C07288=1034.906,183.861,395.226,169.883,42.558,158.045
C07289=1034.912,184.110,395.201,169.886,42.558,158.045
C07290=1034.918,184.359,395.178,169.889,42.558,158.045
C07291=1034.925,184.608,395.155,169.892,42.557,158.046
C07292=1034.930,184.857,395.130,169.895,42.557,158.046
C07293=1034.936,185.105,395.107,169.898,42.556,158.046
C07294=1034.942,185.355,395.082,169.901,42.556,158.046
C07295=1034.948,185.603,395.058,169.904,42.555,158.046
C07296=1034.954,185.852,395.034,169.907,42.555,158.046
C07297=1034.960,186.100,395.010,169.911,42.555,158.046
C07298=1034.966,186.350,394.985,169.914,42.554,158.046
C07299=1034.972,186.598,394.962,169.917,42.554,158.047
C07300=1034.977,186.847,394.937,169.920,42.553,158.047
C07301=1034.984,187.095,394.913,169.923,42.553,158.047
C07302=1034.990,187.344,394.890,169.926,42.552,158.047
C07303=1034.996,187.593,394.865,169.929,42.552,158.047
C07304=1035.002,187.841,394.842,169.932,42.552,158.047
C07305=1035.008,188.091,394.817,169.935,42.552,158.047
C07306=1035.014,188.339,394.793,169.938,42.551,158.048
C07307=1035.021,188.624,394.766,169.941,42.551,158.048
C07308=1035.028,188.907,394.738,169.944,42.550,158.048
C07309=1035.035,189.191,394.710,169.948,42.550,158.048
C07310=1035.041,189.476,394.683,169.952,42.550,158.048
C07311=1035.047,189.724,394.659,169.955,42.549,158.048
C07312=1035.053,189.973,394.635,169.958,42.549,158.048
C07313=1035.059,190.222,394.609,169.962,42.548,158.049
C07314=1035.066,190.470,394.586,169.965,42.548,158.049
C07315=1035.071,190.719,394.561,169.968,42.547,158.049
C07316=1035.077,190.968,394.538,169.971,42.547,158.049
C07317=1035.083,191.217,394.513,169.974,42.547,158.049
C07318=1035.089,191.465,394.489,169.977,42.546,158.049
C07319=1035.095,191.715,394.465,169.980,42.546,158.049
C07320=1035.102,191.964,394.441,169.983,42.545,158.050
C07321=1035.108,192.212,394.416,169.986,42.546,158.050
C07322=1035.114,192.460,394.392,169.989,42.545,158.050
C07323=1035.119,192.709,394.367,169.992,42.545,158.050
C07324=1035.126,192.958,394.343,169.996,42.544,158.050
C07325=1035.132,193.207,394.319,169.999,42.544,158.050
C07326=1035.138,193.455,394.294,170.002,42.544,158.050
C07327=1035.144,193.704,394.270,170.006,42.543,158.051
C07328=1035.151,193.953,394.246,170.009,42.543,158.051
C07329=1035.156,194.202,394.221,170.012,42.542,158.051
C07330=1035.163,194.450,394.197,170.015,42.542,158.051
C07331=1035.169,194.700,394.172,170.018,42.542,158.051
C07332=1035.175,194.948,394.148,170.021,42.541,158.051
C07333=1035.181,195.196,394.123,170.024,42.541,158.051
C07334=1035.188,195.445,394.099,170.027,42.540,158.052
C07335=1035.193,195.694,394.075,170.031,42.541,158.052
C07336=1035.200,195.942,394.050,170.035,42.540,158.052
C07337=1035.206,196.192,394.025,170.038,42.540,158.052
C07338=1035.212,196.440,394.002,170.041,42.539,158.052
C07339=1035.218,196.689,393.976,170.044,42.539,158.052
C07340=1035.224,196.938,393.952,170.047,42.539,158.053
C07341=1035.231,197.187,393.928,170.050,42.538,158.053
C07342=1035.236,197.435,393.903,170.053,42.538,158.053
C07343=1035.243,197.684,393.879,170.057,42.538,158.053
C07344=1035.249,197.932,393.853,170.060,42.537,158.053
C07345=1035.256,198.181,393.829,170.063,42.537,158.053
C07346=1035.262,198.429,393.804,170.067,42.537,158.054
C07347=1035.268,198.678,393.780,170.070,42.536,158.054
C07348=1035.274,198.927,393.755,170.073,42.536,158.054
C07349=1035.281,199.176,393.731,170.077,42.536,158.054
C07350=1035.287,199.425,393.706,170.080,42.536,158.054
C07351=1035.293,199.673,393.682,170.083,42.535,158.054
C07352=1035.299,199.922,393.657,170.086,42.535,158.054
C07353=1035.305,200.171,393.632,170.089,42.535,158.055
C07354=1035.312,200.419,393.607,170.092,42.534,158.055
C07355=1035.318,200.669,393.583,170.096,42.534,158.055
C07356=1035.325,200.916,393.558,170.100,42.534,158.055
C07357=1035.330,201.166,393.534,170.103,42.533,158.055
C07358=1035.337,201.414,393.508,170.106,42.533,158.056
C07359=1035.343,201.663,393.483,170.109,42.533,158.056
C07360=1035.349,201.912,393.458,170.112,42.533,158.056
C07361=1035.354,202.160,393.433,170.116,42.532,158.056
C07362=1035.361,202.409,393.408,170.119,42.533,158.056
C07363=1035.367,202.657,393.383,170.122,42.532,158.057
C07364=1035.373,202.907,393.358,170.126,42.532,158.057
C07365=1035.380,203.155,393.333,170.129,42.532,158.057
C07366=1035.386,203.404,393.308,170.133,42.532,158.057
C07367=1035.391,203.652,393.283,170.136,42.532,158.057
C07368=1035.397,203.901,393.258,170.139,42.532,158.058
C07369=1035.404,204.150,393.233,170.142,42.532,158.058
C07370=1035.410,204.398,393.208,170.145,42.531,158.058
C07371=1035.436,205.448,393.102,170.465,42.636,158.102
C07372=1035.445,205.782,393.066,170.469,42.636,158.102
C07373=1035.454,206.115,393.031,170.472,42.637,158.103
C07374=1035.463,206.448,392.995,170.475,42.638,158.103
C07375=1035.472,206.782,392.960,170.478,42.639,158.104
C07376=1035.479,207.030,392.934,170.480,42.639,158.104
C07377=1035.486,207.279,392.907,170.483,42.640,158.104
C07378=1035.493,207.528,392.881,170.486,42.640,158.105
C07379=1035.499,207.776,392.854,170.488,42.641,158.105
C07380=1035.506,208.025,392.828,170.491,42.641,158.105
C07381=1035.512,208.273,392.802,170.493,42.642,158.105
C07382=1035.519,208.522,392.775,170.495,42.643,158.106
C07383=1035.526,208.771,392.748,170.498,42.644,158.106
C07384=1035.532,209.019,392.722,170.500,42.644,158.106
C07385=1035.540,209.267,392.695,170.502,42.645,158.107
C07386=1035.546,209.516,392.668,170.505,42.645,158.107
C07387=1035.553,209.764,392.642,170.508,42.646,158.107
C07388=1035.560,210.013,392.616,170.510,42.646,158.108
C07389=1035.566,210.262,392.589,170.513,42.647,158.108
C07390=1035.573,210.509,392.562,170.515,42.647,158.108
C07391=1035.580,210.758,392.535,170.517,42.648,158.108
C07392=1035.586,211.007,392.508,170.520,42.649,158.109
C07393=1035.593,211.255,392.482,170.522,42.650,158.109
C07394=1035.600,211.504,392.456,170.524,42.650,158.109
C07395=1035.607,211.752,392.428,170.528,42.651,158.110
C07396=1035.613,212.000,392.402,170.530,42.651,158.110
C07397=1035.620,212.249,392.375,170.532,42.652,158.110
C07398=1035.627,212.497,392.348,170.535,42.653,158.111
C07399=1035.633,212.746,392.321,170.537,42.653,158.111
C07400=1035.639,212.995,392.294,170.539,42.654,158.111
C07401=1035.647,213.243,392.267,170.542,42.654,158.111
C07402=1035.652,213.491,392.240,170.545,42.655,158.112
C07403=1035.660,213.740,392.214,170.547,42.656,158.112
C07404=1035.666,213.989,392.186,170.550,42.656,158.112
C07405=1035.673,214.237,392.160,170.552,42.657,158.113
C07406=1035.679,214.485,392.133,170.554,42.658,158.113
C07407=1035.687,214.734,392.106,170.557,42.659,158.113
C07408=1035.693,214.983,392.079,170.559,42.659,158.114
C07409=1035.700,215.230,392.052,170.562,42.660,158.114
C07410=1035.706,215.479,392.025,170.565,42.660,158.114
C07411=1035.714,215.727,391.998,170.567,42.661,158.115
C07412=1035.719,215.976,391.972,170.569,42.662,158.115
C07413=1035.727,216.224,391.944,170.572,42.662,158.115
C07414=1035.733,216.473,391.917,170.575,42.663,158.116
C07415=1035.741,216.721,391.890,170.577,42.663,158.116
C07416=1035.747,216.970,391.863,170.580,42.664,158.116
C07417=1035.754,217.218,391.836,170.582,42.664,158.116
C07418=1035.760,217.467,391.809,170.584,42.665,158.117
C07419=1035.767,217.715,391.782,170.588,42.666,158.117
C07420=1035.774,217.964,391.755,170.590,42.666,158.117
C07421=1035.781,218.212,391.728,170.593,42.667,158.118
C07422=1035.787,218.460,391.702,170.595,42.668,158.118
C07423=1035.794,218.709,391.674,170.597,42.669,158.118
C07424=1035.801,218.958,391.647,170.600,42.669,158.119
C07425=1035.808,219.206,391.620,170.603,42.670,158.119
C07426=1035.815,219.455,391.593,170.605,42.670,158.119
C07427=1035.821,219.702,391.566,170.608,42.671,158.120
C07428=1035.831,220.042,391.528,170.611,42.672,158.120
C07429=1035.839,220.381,391.492,170.614,42.672,158.120
C07430=1035.848,220.720,391.454,170.618,42.674,158.121
C07431=1035.857,221.059,391.417,170.621,42.675,158.121
C07432=1035.864,221.308,391.390,170.625,42.675,158.122
C07433=1035.870,221.556,391.362,170.627,42.676,158.122
C07434=1035.876,221.804,391.334,170.630,42.677,158.122
C07435=1035.884,222.052,391.307,170.632,42.678,158.123
C07436=1035.890,222.301,391.280,170.635,42.678,158.123
C07437=1035.897,222.550,391.253,170.638,42.679,158.123
C07438=1035.904,222.798,391.225,170.640,42.680,158.124
C07439=1035.910,223.047,391.197,170.642,42.680,158.124
C07440=1035.917,223.296,391.170,170.646,42.681,158.124
C07441=1035.923,223.543,391.143,170.648,42.681,158.125
C07442=1035.930,223.791,391.116,170.650,42.682,158.125
C07443=1035.937,224.040,391.088,170.653,42.683,158.125
C07444=1035.944,224.288,391.060,170.656,42.683,158.126
C07445=1035.950,224.537,391.032,170.659,42.684,158.126
C07446=1035.957,224.786,391.006,170.661,42.685,158.126
C07447=1035.964,225.034,390.978,170.663,42.686,158.127
C07448=1035.971,225.282,390.951,170.667,42.686,158.127
C07449=1035.977,225.531,390.923,170.669,42.687,158.127
C07450=1035.984,225.779,390.895,170.671,42.688,158.128
C07451=1035.990,226.027,390.868,170.675,42.688,158.128
C07452=1035.998,226.275,390.841,170.677,42.689,158.128
C07453=1036.004,226.524,390.813,170.680,42.690,158.129
C07454=1036.011,226.772,390.785,170.682,42.690,158.129
C07455=1036.017,227.021,390.758,170.685,42.691,158.129
C07456=1036.024,227.270,390.730,170.688,42.692,158.130
C07457=1036.031,227.518,390.703,170.690,42.692,158.130
C07458=1036.037,227.766,390.675,170.693,42.693,158.130
C07459=1036.045,228.015,390.648,170.696,42.694,158.131
C07460=1036.051,228.263,390.620,170.698,42.694,158.131
C07461=1036.058,228.511,390.592,170.701,42.695,158.131
C07462=1036.065,228.760,390.565,170.704,42.696,158.132
C07463=1036.071,229.008,390.536,170.706,42.696,158.132
C07464=1036.078,229.256,390.508,170.710,42.697,158.132
C07465=1036.084,229.505,390.480,170.712,42.698,158.133
C07466=1036.091,229.753,390.452,170.714,42.698,158.133
C07467=1036.098,230.002,390.425,170.717,42.699,158.134
C07468=1036.104,230.250,390.397,170.720,42.699,158.134
C07469=1036.111,230.499,390.369,170.722,42.700,158.134
C07470=1036.118,230.747,390.341,170.725,42.701,158.135
C07471=1036.124,230.996,390.314,170.728,42.702,158.135
C07472=1036.131,231.243,390.285,170.731,42.702,158.135
C07473=1036.138,231.492,390.258,170.733,42.703,158.136
C07474=1036.145,231.740,390.230,170.736,42.704,158.136
C07475=1036.151,231.989,390.201,170.739,42.705,158.136
C07476=1036.157,232.237,390.174,170.741,42.706,158.137
C07477=1036.164,232.485,390.145,170.745,42.706,158.137
C07478=1036.171,232.734,390.118,170.747,42.707,158.137
C07479=1036.178,232.982,390.090,170.749,42.708,158.138
C07480=1036.184,233.230,390.061,170.753,42.709,158.138
C07481=1036.191,233.479,390.033,170.755,42.710,158.138
C07482=1036.197,233.727,390.005,170.759,42.710,158.139
C07483=1036.204,233.976,389.978,170.761,42.711,158.139
C07484=1036.213,234.307,389.939,170.765,42.712,158.140
C07485=1036.222,234.639,389.903,170.768,42.713,158.140
C07486=1036.230,234.970,389.864,170.772,42.714,158.141
C07487=1036.240,235.301,389.827,170.776,42.715,158.141
C07488=1036.246,235.550,389.799,170.779,42.716,158.141
C07489=1036.252,235.798,389.771,170.781,42.717,158.142
C07490=1036.259,236.046,389.742,170.784,42.717,158.142
C07491=1036.266,236.295,389.714,170.787,42.718,158.142
C07492=1036.273,236.543,389.686,170.789,42.719,158.143
C07493=1036.279,236.792,389.657,170.793,42.719,158.143
C07494=1036.286,237.040,389.630,170.795,42.720,158.144
C07495=1036.293,237.288,389.601,170.798,42.721,158.144
C07496=1036.300,237.537,389.574,170.801,42.722,158.144
C07497=1036.306,237.785,389.545,170.803,42.723,158.145
C07498=1036.313,238.033,389.517,170.806,42.723,158.145
C07499=1036.320,238.281,389.488,170.809,42.724,158.145
C07500=1036.326,238.530,389.460,170.812,42.725,158.146
C07501=1036.333,238.778,389.431,170.815,42.726,158.146
C07502=1036.340,239.027,389.403,170.818,42.726,158.147
C07503=1036.347,239.275,389.375,170.821,42.727,158.147
C07504=1036.353,239.523,389.347,170.823,42.728,158.147
C07505=1036.360,239.771,389.318,170.826,42.728,158.148
C07506=1036.367,240.020,389.289,170.829,42.729,158.148
C07507=1036.373,240.268,389.261,170.832,42.730,158.148
C07508=1036.380,240.516,389.233,170.835,42.731,158.149
C07509=1036.387,240.765,389.205,170.838,42.732,158.149
C07510=1036.393,241.013,389.176,170.841,42.732,158.150
C07511=1036.400,241.261,389.147,170.843,42.733,158.150
C07512=1036.407,241.509,389.118,170.846,42.734,158.150
C07513=1036.413,241.758,389.090,170.849,42.735,158.151
C07514=1036.420,242.006,389.061,170.852,42.736,158.151
C07515=1036.426,242.254,389.032,170.855,42.737,158.151
C07516=1036.433,242.503,389.005,170.858,42.737,158.152
C07517=1036.440,242.751,388.975,170.861,42.738,158.152
C07518=1036.447,242.999,388.947,170.864,42.739,158.153
C07519=1036.453,243.247,388.918,170.866,42.740,158.153
C07520=1036.459,243.495,388.889,170.869,42.741,158.153
C07521=1036.466,243.744,388.861,170.872,42.742,158.154
C07522=1036.473,243.993,388.831,170.875,42.743,158.154
C07523=1036.480,244.241,388.803,170.878,42.743,158.155
C07524=1036.486,244.489,388.774,170.881,42.744,158.155
C07525=1036.493,244.737,388.746,170.884,42.745,158.155
C07526=1036.499,244.985,388.716,170.887,42.746,158.156
C07527=1036.506,245.234,388.688,170.890,42.747,158.156
C07528=1036.512,245.482,388.659,170.892,42.748,158.157
C07529=1036.518,245.730,388.630,170.896,42.748,158.157
C07530=1036.525,245.978,388.601,170.898,42.749,158.157
C07531=1036.532,246.227,388.572,170.902,42.750,158.158
C07532=1036.538,246.475,388.543,170.904,42.751,158.158
C07533=1036.545,246.723,388.514,170.907,42.752,158.158
C07534=1036.551,246.971,388.485,170.910,42.753,158.159
C07535=1036.558,247.219,388.456,170.913,42.754,158.159
C07536=1036.565,247.468,388.427,170.916,42.755,158.160
C07537=1036.571,247.716,388.398,170.919,42.756,158.160
C07538=1036.578,247.964,388.368,170.922,42.757,158.161
C07539=1036.584,248.213,388.339,170.924,42.757,158.161
C07540=1036.592,248.538,388.301,170.929,42.759,158.162
C07541=1036.601,248.863,388.263,170.933,42.760,158.162
C07542=1036.610,249.189,388.225,170.936,42.761,158.163
C07543=1036.618,249.515,388.186,170.941,42.762,158.163
C07544=1036.626,249.764,388.158,170.943,42.763,158.163
C07545=1036.632,250.012,388.129,170.947,42.764,158.164
C07546=1036.638,250.259,388.099,170.949,42.765,158.164
C07547=1036.645,250.508,388.069,170.953,42.766,158.165
C07548=1036.652,250.756,388.040,170.955,42.767,158.165
C07549=1036.658,251.004,388.011,170.959,42.768,158.166
C07550=1036.665,251.253,387.982,170.961,42.768,158.166
C07551=1036.672,251.501,387.953,170.965,42.769,158.166
C07552=1036.679,251.749,387.923,170.967,42.770,158.167
C07553=1036.685,251.997,387.894,170.971,42.771,158.167
C07554=1036.691,252.245,387.865,170.973,42.772,158.168
C07555=1036.698,252.494,387.836,170.976,42.773,158.168
C07556=1036.705,252.742,387.806,170.980,42.774,158.169
C07557=1036.711,252.990,387.777,170.982,42.775,158.169
C07558=1036.718,253.238,387.748,170.986,42.776,158.169
C07559=1036.725,253.486,387.718,170.988,42.776,158.170
C07560=1036.732,253.735,387.689,170.992,42.778,158.170
C07561=1036.738,253.983,387.660,170.995,42.779,158.171
C07562=1036.745,254.232,387.631,170.998,42.779,158.171
C07563=1036.752,254.479,387.601,171.001,42.780,158.171
C07564=1036.758,254.727,387.572,171.004,42.781,158.172
C07565=1036.765,254.976,387.542,171.007,42.782,158.172
C07566=1036.772,255.223,387.513,171.010,42.783,158.173
C07567=1036.779,255.472,387.484,171.013,42.784,158.173
C07568=1036.785,255.720,387.454,171.017,42.785,158.174
C07569=1036.792,255.969,387.425,171.019,42.786,158.174
C07570=1036.799,256.216,387.395,171.022,42.786,158.174
C07571=1036.806,256.465,387.366,171.026,42.787,158.175
C07572=1036.812,256.713,387.336,171.029,42.789,158.175
C07573=1036.819,256.961,387.306,171.032,42.789,158.176
C07574=1036.826,257.209,387.278,171.034,42.790,158.176
C07575=1036.833,257.457,387.248,171.038,42.791,158.176
C07576=1036.839,257.705,387.219,171.041,42.792,158.177
C07577=1036.847,257.954,387.189,171.044,42.793,158.177
C07578=1036.853,258.202,387.160,171.047,42.794,158.178
C07579=1036.860,258.450,387.129,171.051,42.795,158.178
C07580=1036.867,258.699,387.100,171.053,42.796,158.179
C07581=1036.873,258.946,387.070,171.057,42.796,158.179
C07582=1036.880,259.195,387.041,171.060,42.797,158.179
C07583=1036.887,259.443,387.011,171.063,42.799,158.180
C07584=1036.895,259.691,386.982,171.066,42.799,158.180
C07585=1036.901,259.939,386.953,171.070,42.800,158.181
C07586=1036.908,260.187,386.922,171.072,42.801,158.181
C07587=1036.915,260.436,386.893,171.076,42.802,158.182
C07588=1036.921,260.683,386.863,171.079,42.803,158.182
C07589=1036.929,260.931,386.833,171.083,42.804,158.183
C07590=1036.935,261.180,386.804,171.085,42.805,158.183
C07591=1036.942,261.428,386.774,171.089,42.806,158.183
C07592=1036.949,261.676,386.744,171.092,42.806,158.184
C07593=1036.955,261.924,386.715,171.095,42.808,158.184
C07594=1036.963,262.172,386.685,171.098,42.809,158.185
C07595=1036.969,262.420,386.655,171.102,42.810,158.185
C07596=1036.978,262.745,386.615,171.105,42.811,158.186
C07597=1036.987,263.068,386.576,171.110,42.812,158.186
C07598=1036.996,263.393,386.537,171.114,42.814,158.187
C07599=1037.004,263.718,386.497,171.118,42.815,158.188
C07600=1037.011,263.966,386.467,171.121,42.816,158.188
C07601=1037.017,264.213,386.438,171.125,42.817,158.189
C07602=1037.024,264.462,386.407,171.128,42.818,158.189
C07603=1037.031,264.710,386.377,171.132,42.819,158.189
C07604=1037.037,264.958,386.347,171.134,42.820,158.190
C07605=1037.045,265.206,386.317,171.138,42.822,158.190
C07606=1037.051,265.454,386.286,171.141,42.822,158.191
C07607=1037.058,265.702,386.256,171.144,42.823,158.191
C07608=1037.065,265.950,386.226,171.147,42.825,158.192
C07609=1037.071,266.199,386.196,171.151,42.825,158.192
C07610=1037.078,266.446,386.166,171.154,42.827,158.193
C07611=1037.085,266.694,386.136,171.157,42.828,158.193
C07612=1037.091,266.943,386.105,171.160,42.829,158.194
C07613=1037.098,267.190,386.075,171.164,42.830,158.194
C07614=1037.105,267.438,386.045,171.167,42.830,158.195
C07615=1037.111,267.687,386.014,171.170,42.832,158.195
C07616=1037.118,267.935,385.985,171.173,42.833,158.195
C07617=1037.124,268.183,385.954,171.177,42.834,158.196
C07618=1037.132,268.431,385.924,171.179,42.835,158.196
C07619=1037.138,268.679,385.892,171.183,42.836,158.197
C07620=1037.145,268.927,385.863,171.187,42.838,158.198
C07621=1037.151,269.175,385.832,171.190,42.838,158.198
C07622=1037.158,269.423,385.802,171.194,42.840,158.198
C07623=1037.166,269.672,385.772,171.196,42.840,158.199
C07624=1037.172,269.919,385.741,171.200,42.842,158.199
C07625=1037.179,270.167,385.710,171.203,42.843,158.200
C07626=1037.185,270.416,385.680,171.207,42.844,158.200
C07627=1037.192,270.664,385.650,171.210,42.845,158.201
C07628=1037.199,270.911,385.619,171.213,42.846,158.201
C07629=1037.206,271.159,385.588,171.217,42.847,158.202
C07630=1037.212,271.408,385.558,171.220,42.848,158.202
C07631=1037.219,271.656,385.526,171.224,42.850,158.203
C07632=1037.225,271.903,385.496,171.226,42.850,158.203
C07633=1037.232,272.152,385.466,171.230,42.852,158.204
C07634=1037.239,272.399,385.435,171.233,42.853,158.204
C07635=1037.246,272.648,385.404,171.237,42.854,158.205
C07636=1037.252,272.896,385.373,171.241,42.855,158.205
C07637=1037.259,273.143,385.343,171.243,42.856,158.206
C07638=1037.265,273.392,385.312,171.247,42.857,158.206
C07639=1037.272,273.640,385.281,171.251,42.859,158.207
C07640=1037.279,273.888,385.251,171.254,42.859,158.207
C07641=1037.286,274.136,385.219,171.258,42.861,158.208
C07642=1037.293,274.384,385.189,171.260,42.862,158.208
C07643=1037.299,274.631,385.158,171.264,42.863,158.209
C07644=1037.306,274.880,385.127,171.267,42.864,158.209
C07645=1037.312,275.128,385.096,171.271,42.866,158.210
C07646=1037.320,275.376,385.066,171.275,42.866,158.210
C07647=1037.326,275.624,385.034,171.278,42.868,158.211
C07648=1037.333,275.872,385.003,171.281,42.869,158.211
C07649=1037.340,276.120,384.973,171.284,42.871,158.212
C07650=1037.346,276.367,384.942,171.288,42.871,158.212
C07651=1037.353,276.615,384.910,171.292,42.873,158.213
C07652=1037.362,276.945,384.869,171.296,42.874,158.214
C07653=1037.371,277.273,384.829,171.301,42.876,158.214
C07654=1037.380,277.602,384.787,171.305,42.878,158.215
C07655=1037.389,277.931,384.746,171.310,42.879,158.216
C07656=1037.396,278.179,384.715,171.313,42.880,158.216
C07657=1037.402,278.427,384.684,171.317,42.881,158.217
C07658=1037.409,278.675,384.653,171.321,42.883,158.217
C07659=1037.416,278.922,384.622,171.324,42.884,158.218
C07660=1037.423,279.170,384.590,171.328,42.885,158.218
C07661=1037.429,279.419,384.559,171.330,42.886,158.219
C07662=1037.436,279.667,384.528,171.334,42.888,158.219
C07663=1037.442,279.915,384.496,171.338,42.889,158.220
C07664=1037.449,280.163,384.465,171.341,42.890,158.221
C07665=1037.456,280.411,384.434,171.345,42.892,158.221
C07666=1037.463,280.658,384.402,171.349,42.893,158.222
C07667=1037.469,280.906,384.371,171.352,42.894,158.222
C07668=1037.476,281.154,384.339,171.356,42.896,158.223
C07669=1037.483,281.402,384.308,171.359,42.896,158.223
C07670=1037.489,281.650,384.276,171.362,42.898,158.224
C07671=1037.496,281.898,384.245,171.366,42.899,158.224
C07672=1037.504,282.146,384.214,171.369,42.901,158.225
C07673=1037.510,282.393,384.183,171.373,42.902,158.225
C07674=1037.517,282.641,384.151,171.377,42.903,158.226
C07675=1037.524,282.889,384.120,171.380,42.905,158.227
C07676=1037.531,283.137,384.088,171.384,42.906,158.227
C07677=1037.537,283.385,384.057,171.388,42.907,158.228
C07678=1037.544,283.633,384.026,171.391,42.909,158.228
C07679=1037.551,283.881,383.994,171.395,42.910,158.229
C07680=1037.557,284.129,383.963,171.399,42.911,158.229
C07681=1037.564,284.377,383.931,171.402,42.912,158.230
C07682=1037.571,284.625,383.900,171.406,42.914,158.231
C07683=1037.578,284.872,383.868,171.409,42.915,158.231
C07684=1037.585,285.121,383.837,171.413,42.916,158.232
C07685=1037.592,285.368,383.804,171.417,42.917,158.232
C07686=1037.599,285.616,383.773,171.420,42.919,158.233
C07687=1037.605,285.864,383.742,171.424,42.920,158.233
C07688=1037.612,286.112,383.710,171.428,42.921,158.234
C07689=1037.619,286.360,383.679,171.431,42.922,158.234
C07690=1037.626,286.607,383.647,171.435,42.924,158.235
C07691=1037.633,286.856,383.615,171.439,42.925,158.236
C07692=1037.639,287.104,383.583,171.442,42.926,158.236
C07693=1037.646,287.351,383.551,171.446,42.928,158.237
C07694=1037.653,287.599,383.519,171.450,42.930,158.237
C07695=1037.660,287.847,383.488,171.454,42.931,158.238
C07696=1037.667,288.094,383.456,171.457,42.932,158.239
C07697=1037.673,288.343,383.424,171.461,42.934,158.239
C07698=1037.679,288.591,383.392,171.465,42.935,158.240
C07699=1037.687,288.839,383.360,171.468,42.936,158.240
C07700=1037.694,289.086,383.328,171.472,42.938,158.241
C07701=1037.701,289.334,383.296,171.476,42.939,158.241
C07702=1037.707,289.582,383.264,171.479,42.941,158.242
C07703=1037.714,289.829,383.232,171.483,42.942,158.243
C07704=1037.721,290.078,383.200,171.487,42.944,158.243
C07705=1037.728,290.325,383.167,171.490,42.945,158.244
C07706=1037.734,290.573,383.136,171.494,42.946,158.244
C07707=1037.741,290.821,383.104,171.498,42.948,158.245
C07708=1037.751,291.162,383.060,171.503,42.950,158.246
C07709=1037.760,291.503,383.015,171.508,42.952,158.247
C07710=1037.769,291.843,382.971,171.513,42.954,158.248
C07711=1037.779,292.185,382.927,171.519,42.956,158.248
C07712=1037.786,292.432,382.895,171.522,42.957,158.249
C07713=1037.792,292.681,382.863,171.526,42.959,158.250
C07714=1037.799,292.928,382.830,171.530,42.960,158.250
C07715=1037.806,293.175,382.798,171.534,42.961,158.251
C07716=1037.813,293.423,382.766,171.537,42.963,158.251
C07717=1037.820,293.672,382.734,171.541,42.965,158.252
C07718=1037.827,293.919,382.702,171.545,42.966,158.253
C07719=1037.833,294.166,382.669,171.548,42.967,158.253
C07720=1037.841,294.414,382.636,171.552,42.969,158.254
C07721=1037.847,294.663,382.604,171.556,42.971,158.254
C07722=1037.854,294.910,382.572,171.561,42.972,158.255
C07723=1037.861,295.158,382.539,171.565,42.974,158.256
C07724=1037.868,295.405,382.507,171.568,42.975,158.256
C07725=1037.874,295.653,382.474,171.572,42.977,158.257
C07726=1037.881,295.901,382.441,171.576,42.978,158.258
C07727=1037.887,296.149,382.408,171.580,42.980,158.258
C07728=1037.894,296.396,382.376,171.583,42.981,158.259
C07729=1037.901,296.644,382.343,171.587,42.983,158.260
C07730=1037.908,296.892,382.310,171.591,42.985,158.260
C07731=1037.914,297.140,382.278,171.595,42.987,158.261
C07732=1037.921,297.387,382.245,171.598,42.988,158.262
C07733=1037.928,297.635,382.212,171.602,42.990,158.262
C07734=1037.934,297.883,382.180,171.607,42.991,158.263
C07735=1037.940,298.130,382.147,171.611,42.993,158.264
C07736=1037.948,298.378,382.114,171.615,42.994,158.264
C07737=1037.954,298.626,382.082,171.618,42.996,158.265
C07738=1037.961,298.873,382.048,171.622,42.997,158.265
C07739=1037.968,299.121,382.015,171.626,42.999,158.266
C07740=1037.975,299.369,381.983,171.630,43.001,158.267
C07741=1037.982,299.617,381.950,171.635,43.002,158.268
C07742=1037.988,299.864,381.917,171.638,43.004,158.268
C07743=1037.995,300.113,381.884,171.642,43.006,158.269
C07744=1038.002,300.359,381.851,171.646,43.008,158.270
C07745=1038.009,300.607,381.818,171.650,43.009,158.270
C07746=1038.015,300.855,381.785,171.653,43.011,158.271
C07747=1038.022,301.103,381.752,171.657,43.013,158.272
C07748=1038.029,301.351,381.719,171.662,43.014,158.272
C07749=1038.036,301.598,381.687,171.666,43.016,158.273
C07750=1038.043,301.846,381.653,171.670,43.018,158.274
C07751=1038.050,302.093,381.620,171.673,43.019,158.274
C07752=1038.056,302.341,381.587,171.677,43.021,158.275
C07753=1038.063,302.589,381.555,171.682,43.023,158.276
C07754=1038.071,302.836,381.521,171.686,43.024,158.276
C07755=1038.077,303.084,381.488,171.690,43.026,158.277
C07756=1038.084,303.332,381.454,171.694,43.028,158.278
C07757=1038.090,303.579,381.422,171.698,43.029,158.278
C07758=1038.098,303.827,381.389,171.702,43.031,158.279
C07759=1038.105,304.075,381.355,171.706,43.033,158.280
C07760=1038.112,304.322,381.322,171.710,43.034,158.280
C07761=1038.119,304.570,381.289,171.714,43.036,158.281
C07762=1038.125,304.818,381.256,171.719,43.038,158.282
C07763=1038.133,305.065,381.223,171.722,43.040,158.283
C07764=1038.139,305.284,381.194,171.726,43.041,158.283
C07765=1038.145,305.503,381.164,171.730,43.042,158.284
C07766=1038.151,305.721,381.135,171.733,43.043,158.284
C07767=1038.157,305.940,381.106,171.737,43.045,158.285
C07768=1038.168,306.326,381.053,171.744,43.048,158.286
C07769=1038.179,306.713,381.001,171.750,43.051,158.287
C07770=1038.190,307.099,380.949,171.756,43.053,158.288
C07771=1038.201,307.486,380.897,171.762,43.056,158.289
C07772=1038.208,307.734,380.864,171.766,43.058,158.290
C07773=1038.216,307.981,380.831,171.771,43.059,158.291
C07774=1038.222,308.228,380.797,171.775,43.061,158.292
C07775=1038.229,308.476,380.763,171.779,43.063,158.292
C07776=1038.236,308.724,380.730,171.784,43.064,158.293
C07777=1038.244,308.972,380.696,171.788,43.066,158.294
C07778=1038.250,309.219,380.663,171.791,43.068,158.294
C07779=1038.258,309.466,380.630,171.796,43.070,158.295
C07780=1038.265,309.715,380.597,171.800,43.072,158.296
C07781=1038.272,309.962,380.563,171.804,43.074,158.297
C07782=1038.279,310.209,380.529,171.809,43.075,158.297
C07783=1038.286,310.457,380.495,171.813,43.077,158.298
C07784=1038.293,310.705,380.462,171.817,43.079,158.299
C07785=1038.301,310.952,380.428,171.821,43.080,158.299
C07786=1038.308,311.200,380.395,171.825,43.082,158.300
C07787=1038.315,311.448,380.361,171.830,43.084,158.301
C07788=1038.322,311.696,380.328,171.834,43.086,158.302
C07789=1038.329,311.943,380.294,171.838,43.088,158.302
C07790=1038.336,312.190,380.260,171.843,43.089,158.303
C07791=1038.343,312.438,380.226,171.847,43.091,158.304
C07792=1038.350,312.685,380.191,171.851,43.094,158.305
C07793=1038.356,312.933,380.157,171.856,43.096,158.305
C07794=1038.363,313.180,380.123,171.860,43.097,158.306
C07795=1038.370,313.428,380.090,171.864,43.099,158.307
C07796=1038.377,313.676,380.055,171.869,43.101,158.308
C07797=1038.384,313.923,380.021,171.873,43.104,158.309
C07798=1038.390,314.170,379.987,171.877,43.105,158.309
C07799=1038.397,314.418,379.953,171.881,43.107,158.310
C07800=1038.404,314.666,379.918,171.885,43.109,158.311
C07801=1038.411,314.913,379.884,171.890,43.111,158.312
C07802=1038.418,315.161,379.849,171.894,43.113,158.312
C07803=1038.425,315.409,379.816,171.898,43.115,158.313
C07804=1038.433,315.656,379.781,171.903,43.117,158.314
C07805=1038.439,315.904,379.747,171.907,43.119,158.315
C07806=1038.446,316.151,379.713,171.912,43.121,158.316
C07807=1038.452,316.398,379.678,171.916,43.124,158.317
C07808=1038.460,316.646,379.644,171.920,43.125,158.317
C07809=1038.466,316.893,379.609,171.925,43.127,158.318
C07810=1038.474,317.141,379.575,171.929,43.130,158.319
C07811=1038.480,317.388,379.540,171.934,43.131,158.320
C07812=1038.488,317.636,379.506,171.938,43.133,158.320
C07813=1038.494,317.883,379.471,171.943,43.136,158.321
C07814=1038.502,318.131,379.437,171.947,43.137,158.322
C07815=1038.509,318.378,379.403,171.951,43.139,158.323
C07816=1038.515,318.626,379.368,171.956,43.142,158.324
C07817=1038.523,318.873,379.334,171.960,43.143,158.324
C07818=1038.529,319.121,379.299,171.965,43.146,158.325
C07819=1038.537,319.368,379.265,171.969,43.148,158.326
C07820=1038.547,319.731,379.214,171.975,43.151,158.327
C07821=1038.557,320.093,379.164,171.982,43.154,158.329
C07822=1038.568,320.455,379.113,171.989,43.157,158.330
C07823=1038.578,320.818,379.062,171.996,43.160,158.331
C07824=1038.586,321.065,379.028,172.000,43.162,158.332
C07825=1038.592,321.312,378.992,172.005,43.164,158.333
C07826=1038.600,321.560,378.959,172.009,43.166,158.334
C07827=1038.606,321.807,378.923,172.014,43.168,158.334
C07828=1038.614,322.055,378.889,172.018,43.170,158.335
C07829=1038.621,322.302,378.853,172.023,43.172,158.336
C07830=1038.628,322.550,378.820,172.027,43.175,158.337
C07831=1038.635,322.797,378.784,172.032,43.177,158.338
C07832=1038.643,323.044,378.750,172.036,43.179,158.339
C07833=1038.649,323.292,378.715,172.041,43.181,158.339
C07834=1038.658,323.540,378.680,172.046,43.183,158.340
C07835=1038.664,323.787,378.645,172.050,43.185,158.341
C07836=1038.671,324.035,378.610,172.055,43.188,158.342
C07837=1038.678,324.282,378.576,172.059,43.189,158.343
C07838=1038.686,324.530,378.540,172.064,43.192,158.344
C07839=1038.693,324.777,378.506,172.068,43.194,158.344
C07840=1038.700,325.025,378.471,172.073,43.196,158.345
C07841=1038.708,325.272,378.436,172.078,43.198,158.346
C07842=1038.715,325.520,378.401,172.082,43.200,158.347
C07843=1038.722,325.767,378.366,172.087,43.202,158.348
C07844=1038.730,326.015,378.330,172.092,43.205,158.349
C07845=1038.737,326.262,378.296,172.097,43.207,158.350
C07846=1038.744,326.509,378.261,172.102,43.209,158.351
C07847=1038.752,326.757,378.226,172.106,43.211,158.351
C07848=1038.759,327.004,378.191,172.111,43.214,158.352
C07849=1038.766,327.251,378.155,172.116,43.216,158.353
C07850=1038.774,327.499,378.120,172.120,43.218,158.354
C07851=1038.781,327.746,378.085,172.125,43.220,158.355
C07852=1038.789,327.994,378.050,172.130,43.222,158.356
C07853=1038.796,328.241,378.015,172.134,43.225,158.357
C07854=1038.803,328.488,377.980,172.139,43.226,158.358
C07855=1038.811,328.736,377.944,172.144,43.229,158.359
C07856=1038.818,328.983,377.909,172.148,43.231,158.359
C07857=1038.825,329.231,377.873,172.154,43.233,158.360
C07858=1038.832,329.478,377.838,172.159,43.236,158.361
C07859=1038.839,329.725,377.802,172.163,43.238,158.362
C07860=1038.847,329.973,377.766,172.168,43.241,158.363
C07861=1038.853,330.220,377.731,172.173,43.243,158.364
C07862=1038.861,330.468,377.695,172.177,43.245,158.365
C07863=1038.868,330.715,377.660,172.182,43.248,158.366
C07864=1038.875,330.962,377.624,172.188,43.250,158.367
C07865=1038.882,331.210,377.588,172.192,43.253,158.368
C07866=1038.890,331.457,377.552,172.197,43.255,158.369
C07867=1038.897,331.705,377.517,172.202,43.257,158.370
C07868=1038.904,331.952,377.481,172.206,43.260,158.371
C07869=1038.911,332.199,377.446,172.211,43.262,158.372
C07870=1038.919,332.447,377.409,172.216,43.264,158.372
C07871=1038.927,332.693,377.374,172.221,43.267,158.373
C07872=1038.934,332.941,377.339,172.226,43.270,158.374
C07873=1038.941,333.188,377.303,172.231,43.272,158.375
C07874=1038.949,333.435,377.267,172.236,43.274,158.376
C07875=1038.955,333.683,377.232,172.240,43.277,158.377
C07876=1038.966,334.041,377.180,172.248,43.280,158.379
C07877=1038.977,334.398,377.128,172.255,43.284,158.380
C07878=1038.987,334.756,377.076,172.263,43.287,158.382
C07879=1038.998,335.114,377.024,172.269,43.291,158.383
C07880=1039.006,335.361,376.987,172.274,43.294,158.384
C07881=1039.012,335.608,376.951,172.280,43.296,158.385
C07882=1039.020,335.856,376.915,172.284,43.299,158.386
C07883=1039.027,336.103,376.879,172.289,43.301,158.387
C07884=1039.034,336.350,376.843,172.294,43.304,158.388
C07885=1039.041,336.597,376.806,172.300,43.306,158.389
C07886=1039.048,336.844,376.770,172.305,43.309,158.390
C07887=1039.056,337.092,376.734,172.309,43.312,158.391
C07888=1039.064,337.339,376.698,172.314,43.314,158.392
C07889=1039.071,337.587,376.661,172.320,43.317,158.393
C07890=1039.078,337.834,376.625,172.325,43.319,158.394
C07891=1039.085,338.081,376.589,172.330,43.322,158.395
C07892=1039.093,338.328,376.552,172.334,43.324,158.396
C07893=1039.100,338.575,376.515,172.340,43.327,158.397
C07894=1039.107,338.822,376.479,172.345,43.330,158.398
C07895=1039.115,339.070,376.443,172.350,43.332,158.399
C07896=1039.123,339.317,376.407,172.356,43.335,158.400
C07897=1039.129,339.564,376.370,172.361,43.337,158.401
C07898=1039.137,339.811,376.333,172.366,43.340,158.402
C07899=1039.145,340.059,376.297,172.370,43.343,158.403
C07900=1039.152,340.306,376.261,172.376,43.345,158.404
C07901=1039.160,340.553,376.223,172.381,43.348,158.405
C07902=1039.167,340.801,376.187,172.386,43.351,158.406
C07903=1039.174,341.047,376.151,172.391,43.353,158.407
C07904=1039.182,341.294,376.114,172.397,43.356,158.408
C07905=1039.189,341.542,376.078,172.402,43.359,158.409
C07906=1039.197,341.789,376.041,172.407,43.361,158.410
C07907=1039.204,342.037,376.004,172.413,43.364,158.411
C07908=1039.212,342.284,375.968,172.417,43.367,158.413
C07909=1039.219,342.531,375.930,172.422,43.370,158.414
C07910=1039.227,342.777,375.894,172.428,43.373,158.415
C07911=1039.234,343.025,375.857,172.433,43.375,158.416
C07912=1039.242,343.272,375.820,172.438,43.378,158.417
C07913=1039.248,343.520,375.783,172.444,43.381,158.418
C07914=1039.256,343.766,375.746,172.449,43.384,158.419
C07915=1039.264,344.014,375.709,172.454,43.386,158.420
C07916=1039.271,344.261,375.672,172.460,43.389,158.421
C07917=1039.279,344.508,375.635,172.465,43.392,158.422
C07918=1039.287,344.755,375.598,172.471,43.395,158.423
C07919=1039.294,345.003,375.561,172.476,43.398,158.425
C07920=1039.301,345.250,375.523,172.481,43.401,158.426
C07921=1039.309,345.497,375.487,172.487,43.403,158.427
C07922=1039.316,345.744,375.449,172.492,43.406,158.428
C07923=1039.324,345.991,375.412,172.497,43.409,158.429
C07924=1039.331,346.238,375.375,172.503,43.412,158.430
C07925=1039.338,346.486,375.338,172.508,43.415,158.431
C07926=1039.346,346.732,375.301,172.514,43.418,158.432
C07927=1039.353,346.979,375.263,172.519,43.421,158.434
C07928=1039.361,347.226,375.226,172.525,43.424,158.435
C07929=1039.369,347.473,375.189,172.530,43.427,158.436
C07930=1039.376,347.721,375.151,172.535,43.430,158.437
C07931=1039.384,347.967,375.114,172.541,43.432,158.438
C07932=1039.395,348.322,375.061,172.549,43.437,158.440
C07933=1039.406,348.676,375.007,172.557,43.441,158.441
C07934=1039.417,349.030,374.953,172.564,43.445,158.443
C07935=1039.427,349.384,374.900,172.572,43.449,158.445
C07936=1039.435,349.631,374.863,172.577,43.452,158.446
C07937=1039.443,349.877,374.824,172.583,43.456,158.447
C07938=1039.451,350.125,374.787,172.588,43.458,158.448
C07939=1039.458,350.372,374.749,172.595,43.462,158.449
C07940=1039.465,350.619,374.712,172.600,43.464,158.450
C07941=1039.473,350.866,374.674,172.606,43.467,158.452
C07942=1039.481,351.113,374.636,172.611,43.471,158.453
C07943=1039.488,351.361,374.598,172.617,43.474,158.454
C07944=1039.496,351.607,374.560,172.622,43.477,158.455
C07945=1039.503,351.854,374.523,172.628,43.480,158.456
C07946=1039.511,352.101,374.484,172.633,43.483,158.458
C07947=1039.519,352.349,374.447,172.639,43.487,158.459
C07948=1039.526,352.596,374.409,172.645,43.489,158.460
C07949=1039.533,352.842,374.371,172.651,43.493,158.461
C07950=1039.541,353.089,374.334,172.656,43.495,158.462
C07951=1039.549,353.336,374.295,172.662,43.499,158.464
C07952=1039.557,353.583,374.257,172.668,43.502,158.465
C07953=1039.564,353.830,374.219,172.673,43.505,158.466
C07954=1039.572,354.077,374.181,172.680,43.508,158.467
C07955=1039.580,354.324,374.143,172.685,43.512,158.469
C07956=1039.588,354.572,374.105,172.691,43.514,158.470
C07957=1039.595,354.818,374.066,172.696,43.518,158.471
C07958=1039.603,355.065,374.029,172.702,43.521,158.472
C07959=1039.611,355.312,373.990,172.709,43.524,158.474
C07960=1039.618,355.559,373.952,172.714,43.527,158.475
C07961=1039.627,355.806,373.914,172.720,43.530,158.476
C07962=1039.634,356.053,373.877,172.725,43.534,158.477
C07963=1039.643,356.300,373.838,172.732,43.537,158.479
C07964=1039.650,356.547,373.800,172.737,43.540,158.480
C07965=1039.658,356.793,373.761,172.743,43.544,158.481
C07966=1039.665,357.041,373.722,172.749,43.547,158.482
C07967=1039.673,357.287,373.684,172.755,43.550,158.484
C07968=1039.681,357.534,373.645,172.761,43.553,158.485
C07969=1039.688,357.781,373.607,172.766,43.557,158.486
C07970=1039.697,358.028,373.569,172.773,43.560,158.487
C07971=1039.704,358.275,373.530,172.779,43.564,158.489
C07972=1039.712,358.522,373.492,172.785,43.567,158.490
C07973=1039.720,358.768,373.453,172.790,43.570,158.491
C07974=1039.728,359.016,373.415,172.797,43.574,158.493
C07975=1039.735,359.263,373.376,172.802,43.577,158.494
C07976=1039.743,359.510,373.337,172.808,43.580,158.495
C07977=1039.751,359.757,373.299,172.815,43.584,158.497
C07978=1039.759,360.003,373.260,172.820,43.587,158.498
C07979=1039.767,360.250,373.221,172.826,43.591,158.499
C07980=1039.775,360.497,373.183,172.833,43.594,158.501
C07981=1039.783,360.744,373.144,172.838,43.597,158.502
C07982=1039.790,360.991,373.104,172.844,43.601,158.503
C07983=1039.799,361.238,373.066,172.851,43.605,158.505
C07984=1039.806,361.484,373.028,172.857,43.608,158.506
C07985=1039.815,361.731,372.988,172.863,43.611,158.507
C07986=1039.823,361.978,372.950,172.869,43.614,158.509
C07987=1039.830,362.224,372.910,172.875,43.618,158.510
C07988=1039.841,362.585,372.854,172.884,43.623,158.512
C07989=1039.853,362.945,372.797,172.893,43.629,158.514
C07990=1039.864,363.306,372.739,172.903,43.634,158.516
C07991=1039.876,363.666,372.682,172.911,43.639,158.518
C07992=1039.884,363.912,372.643,172.918,43.642,158.519
C07993=1039.891,364.159,372.603,172.924,43.646,158.521
C07994=1039.900,364.405,372.564,172.929,43.650,158.522
C07995=1039.907,364.653,372.524,172.936,43.653,158.524
C07996=1039.916,364.899,372.485,172.942,43.657,158.525
C07997=1039.923,365.145,372.446,172.949,43.661,158.526
C07998=1039.931,365.392,372.406,172.955,43.664,158.528
C07999=1039.939,365.639,372.368,172.961,43.668,158.529
C08000=1039.947,365.886,372.328,172.967,43.672,158.531
C08001=1039.956,366.133,372.288,172.974,43.675,158.532
C08002=1039.963,366.380,372.248,172.980,43.679,158.534
C08003=1039.972,366.626,372.209,172.987,43.683,158.535
C08004=1039.979,366.872,372.170,172.993,43.687,158.537
C08005=1039.987,367.119,372.130,173.000,43.691,158.538
C08006=1039.995,367.366,372.090,173.006,43.694,158.539
C08007=1040.003,367.613,372.051,173.012,43.698,158.541
C08008=1040.011,367.859,372.011,173.019,43.701,158.542
C08009=1040.020,368.106,371.972,173.025,43.705,158.544
C08010=1040.027,368.353,371.932,173.032,43.709,158.545
C08011=1040.036,368.600,371.893,173.038,43.713,158.547
C08012=1040.044,368.846,371.853,173.045,43.717,158.548
C08013=1040.052,369.092,371.813,173.051,43.720,158.550
C08014=1040.061,369.339,371.773,173.057,43.724,158.551
C08015=1040.068,369.586,371.733,173.064,43.728,158.553
C08016=1040.078,369.833,371.694,173.070,43.732,158.554
C08017=1040.085,370.080,371.654,173.077,43.736,158.556
C08018=1040.093,370.326,371.613,173.084,43.739,158.557
C08019=1040.102,370.573,371.574,173.090,43.744,158.559
C08020=1040.110,370.819,371.533,173.097,43.747,158.560
C08021=1040.117,371.066,371.493,173.104,43.751,158.562
C08022=1040.125,371.313,371.453,173.110,43.756,158.563
C08023=1040.134,371.559,371.413,173.117,43.759,158.565
C08024=1040.142,371.805,371.373,173.124,43.763,158.566
C08025=1040.150,372.052,371.333,173.130,43.768,158.568
C08026=1040.158,372.299,371.292,173.137,43.771,158.570
C08027=1040.166,372.546,371.252,173.144,43.775,158.571
C08028=1040.175,372.792,371.212,173.150,43.779,158.573
C08029=1040.183,373.038,371.171,173.157,43.783,158.574
C08030=1040.191,373.285,371.131,173.164,43.787,158.576
C08031=1040.199,373.532,371.091,173.171,43.791,158.577
C08032=1040.207,373.779,371.050,173.177,43.796,158.579
C08033=1040.215,374.025,371.009,173.184,43.799,158.580
C08034=1040.224,374.271,370.970,173.191,43.804,158.582
C08035=1040.232,374.518,370.929,173.198,43.808,158.584
C08036=1040.240,374.765,370.888,173.204,43.812,158.585
C08037=1040.248,375.011,370.847,173.211,43.816,158.587
C08038=1040.256,375.257,370.807,173.218,43.820,158.589
C08039=1040.265,375.504,370.766,173.225,43.824,158.590
C08040=1040.274,375.750,370.726,173.233,43.828,158.592
C08041=1040.282,375.997,370.685,173.239,43.833,158.593
C08042=1040.290,376.244,370.644,173.246,43.837,158.595
C08043=1040.298,376.490,370.603,173.253,43.841,158.597
C08044=1040.311,376.870,370.541,173.264,43.847,158.599
C08045=1040.324,377.250,370.477,173.274,43.854,158.602
C08046=1040.338,377.630,370.415,173.286,43.860,158.604
C08047=1040.351,378.010,370.352,173.296,43.867,158.607
C08048=1040.359,378.257,370.311,173.303,43.871,158.608
C08049=1040.368,378.503,370.269,173.310,43.875,158.610
C08050=1040.376,378.749,370.229,173.317,43.879,158.612
C08051=1040.385,378.996,370.188,173.325,43.884,158.613
C08052=1040.393,379.242,370.146,173.332,43.888,158.615
C08053=1040.402,379.489,370.105,173.339,43.893,158.617
C08054=1040.409,379.735,370.064,173.346,43.897,158.619
C08055=1040.418,379.982,370.022,173.353,43.901,158.620
C08056=1040.426,380.228,369.981,173.360,43.906,158.622
C08057=1040.435,380.475,369.940,173.367,43.910,158.624
C08058=1040.443,380.720,369.899,173.374,43.915,158.626
C08059=1040.451,380.967,369.856,173.382,43.919,158.627
C08060=1040.460,381.214,369.815,173.389,43.924,158.629
C08061=1040.468,381.460,369.774,173.396,43.928,158.631
C08062=1040.477,381.706,369.732,173.403,43.933,158.633
C08063=1040.486,381.953,369.691,173.411,43.937,158.634
C08064=1040.493,382.199,369.649,173.418,43.942,158.636
C08065=1040.502,382.445,369.608,173.425,43.946,158.638
C08066=1040.511,382.692,369.566,173.433,43.951,158.640
C08067=1040.520,382.937,369.525,173.440,43.955,158.642
C08068=1040.528,383.184,369.483,173.448,43.959,158.643
C08069=1040.537,383.430,369.441,173.456,43.964,158.645
C08070=1040.546,383.677,369.399,173.463,43.969,158.647
C08071=1040.554,383.923,369.358,173.470,43.973,158.649
C08072=1040.563,384.169,369.316,173.478,43.978,158.650
C08073=1040.572,384.415,369.274,173.485,43.983,158.652
C08074=1040.580,384.662,369.232,173.493,43.988,158.654
C08075=1040.589,384.908,369.190,173.500,43.992,158.656
C08076=1040.597,385.154,369.149,173.507,43.997,158.658
C08077=1040.606,385.400,369.107,173.516,44.001,158.660
C08078=1040.614,385.647,369.065,173.523,44.006,158.661
C08079=1040.623,385.893,369.023,173.531,44.011,158.663
C08080=1040.633,386.139,368.981,173.538,44.015,158.665
C08081=1040.642,386.385,368.939,173.545,44.020,158.667
C08082=1040.650,386.632,368.897,173.554,44.025,158.669
C08083=1040.659,386.878,368.855,173.561,44.029,158.671
C08084=1040.668,387.124,368.812,173.569,44.034,158.673
C08085=1040.677,387.370,368.771,173.576,44.039,158.675
C08086=1040.685,387.617,368.728,173.585,44.044,158.676
C08087=1040.694,387.863,368.686,173.592,44.048,158.678
C08088=1040.704,388.109,368.644,173.600,44.054,158.680
C08089=1040.712,388.355,368.601,173.607,44.058,158.682
C08090=1040.721,388.601,368.559,173.616,44.063,158.684
C08091=1040.729,388.848,368.516,173.623,44.068,158.686
C08092=1040.738,389.093,368.474,173.631,44.073,158.688
C08093=1040.747,389.339,368.431,173.639,44.078,158.690
C08094=1040.756,389.585,368.389,173.647,44.083,158.692
C08095=1040.764,389.832,368.346,173.654,44.088,158.694
C08096=1040.774,390.078,368.303,173.663,44.093,158.696
C08097=1040.783,390.324,368.260,173.671,44.097,158.698
C08098=1040.792,390.570,368.218,173.678,44.103,158.700
C08099=1040.800,390.816,368.175,173.687,44.107,158.702
C08100=1040.816,391.230,368.104,173.700,44.116,158.705
C08101=1040.830,391.645,368.031,173.714,44.124,158.708
C08102=1040.846,392.058,367.959,173.727,44.133,158.712
C08103=1040.861,392.472,367.886,173.741,44.142,158.715
C08104=1040.869,392.718,367.843,173.750,44.147,158.717
C08105=1040.879,392.964,367.801,173.757,44.152,158.720
C08106=1040.888,393.211,367.757,173.765,44.157,158.722
C08107=1040.896,393.457,367.714,173.774,44.163,158.724
C08108=1040.906,393.702,367.671,173.781,44.168,158.726
C08109=1040.915,393.949,367.628,173.790,44.173,158.728
C08110=1040.923,394.195,367.585,173.798,44.178,158.730
C08111=1040.934,394.441,367.541,173.807,44.183,158.732
C08112=1040.942,394.687,367.498,173.815,44.188,158.734
C08113=1040.951,394.932,367.454,173.823,44.194,158.736
C08114=1040.960,395.179,367.411,173.832,44.199,158.738
C08115=1040.970,395.424,367.368,173.840,44.204,158.740
C08116=1040.979,395.671,367.325,173.848,44.209,158.742
C08117=1040.987,395.916,367.281,173.856,44.215,158.744
C08118=1040.997,396.162,367.237,173.865,44.220,158.747
C08119=1041.005,396.409,367.194,173.874,44.225,158.749
C08120=1041.015,396.655,367.150,173.882,44.231,158.751
C08121=1041.024,396.900,367.106,173.891,44.236,158.753
C08122=1041.034,397.146,367.062,173.900,44.242,158.755
C08123=1041.042,397.392,367.019,173.907,44.247,158.757
C08124=1041.052,397.638,366.975,173.916,44.253,158.760
C08125=1041.061,397.884,366.931,173.925,44.258,158.762
C08126=1041.070,398.130,366.887,173.933,44.264,158.764
C08127=1041.079,398.376,366.843,173.942,44.269,158.766
C08128=1041.089,398.622,366.799,173.951,44.275,158.769
C08129=1041.097,398.867,366.755,173.960,44.280,158.771
C08130=1041.107,399.114,366.711,173.968,44.286,158.773
C08131=1041.117,399.359,366.668,173.977,44.291,158.775
C08132=1041.126,399.605,366.624,173.986,44.297,158.778
C08133=1041.136,399.850,366.579,173.995,44.302,158.780
C08134=1041.145,400.096,366.535,174.003,44.308,158.782
C08135=1041.154,400.343,366.491,174.012,44.314,158.784
C08136=1041.164,400.589,366.447,174.021,44.319,158.787
C08137=1041.174,400.834,366.402,174.030,44.325,158.789
C08138=1041.182,401.080,366.358,174.039,44.330,158.791
C08139=1041.192,401.326,366.314,174.048,44.337,158.794
C08140=1041.201,401.571,366.269,174.056,44.342,158.796
C08141=1041.210,401.818,366.225,174.065,44.348,158.798
C08142=1041.220,402.063,366.180,174.075,44.354,158.801
C08143=1041.229,402.309,366.136,174.084,44.360,158.803
C08144=1041.239,402.555,366.091,174.093,44.365,158.805
C08145=1041.249,402.800,366.046,174.102,44.371,158.808
C08146=1041.258,403.047,366.002,174.111,44.377,158.810
C08147=1041.267,403.292,365.956,174.120,44.383,158.812
C08148=1041.277,403.538,365.912,174.129,44.388,158.815
C08149=1041.286,403.783,365.867,174.139,44.395,158.817
C08150=1041.296,404.030,365.823,174.148,44.401,158.820
C08151=1041.305,404.275,365.777,174.157,44.406,158.822
C08152=1041.315,404.521,365.732,174.166,44.412,158.824
C08153=1041.324,404.766,365.688,174.176,44.418,158.827
C08154=1041.333,405.012,365.642,174.185,44.424,158.829
C08155=1041.343,405.258,365.597,174.194,44.431,158.832
C08156=1041.352,405.475,365.557,174.202,44.436,158.834
C08157=1041.360,405.692,365.517,174.211,44.441,158.836
C08158=1041.369,405.909,365.477,174.219,44.446,158.838
C08159=1041.377,406.126,365.438,174.227,44.452,158.840
C08160=1041.386,406.342,365.397,174.236,44.457,158.843
C08161=1041.394,406.559,365.357,174.244,44.463,158.845
C08162=1041.403,406.776,365.317,174.253,44.468,158.847
C08163=1041.411,406.993,365.277,174.261,44.473,158.849
C08164=1041.421,407.238,365.233,174.270,44.479,158.852
C08165=1041.431,407.484,365.187,174.279,44.486,158.854
C08166=1041.440,407.730,365.141,174.290,44.492,158.857
C08167=1041.451,407.975,365.095,174.299,44.498,158.859
C08168=1041.460,408.221,365.050,174.308,44.504,158.862
C08169=1041.470,408.466,365.004,174.318,44.511,158.864
C08170=1041.480,408.712,364.959,174.327,44.517,158.867
C08171=1041.489,408.957,364.913,174.338,44.523,158.870
C08172=1041.500,409.204,364.868,174.347,44.529,158.872
C08173=1041.510,409.449,364.822,174.357,44.536,158.875
C08174=1041.520,409.695,364.776,174.368,44.542,158.877
C08175=1041.529,409.940,364.731,174.377,44.548,158.880
C08176=1041.539,410.186,364.685,174.386,44.555,158.883
C08177=1041.550,410.432,364.639,174.397,44.561,158.885
C08178=1041.560,410.676,364.593,174.407,44.568,158.888
C08179=1041.569,410.923,364.547,174.417,44.573,158.890
C08180=1041.579,411.168,364.502,174.427,44.580,158.893
C08181=1041.589,411.414,364.455,174.436,44.587,158.896
C08182=1041.600,411.659,364.409,174.447,44.593,158.898
C08183=1041.610,411.905,364.363,174.456,44.599,158.901
C08184=1041.620,412.150,364.317,174.467,44.606,158.904
C08185=1041.630,412.395,364.270,174.477,44.613,158.907
C08186=1041.640,412.641,364.224,174.488,44.619,158.909
C08187=1041.650,412.886,364.178,174.497,44.626,158.912
C08188=1041.660,413.132,364.132,174.508,44.633,158.915
C08189=1041.670,413.377,364.084,174.518,44.639,158.918
C08190=1041.680,413.623,364.038,174.529,44.646,158.921
C08191=1041.691,413.868,363.991,174.539,44.652,158.923
C08192=1041.700,414.113,363.945,174.549,44.660,158.926
C08193=1041.710,414.359,363.898,174.560,44.666,158.929
C08194=1041.720,414.605,363.851,174.570,44.673,158.932
C08195=1041.731,414.850,363.805,174.581,44.680,158.935
C08196=1041.741,415.096,363.758,174.591,44.686,158.937
C08197=1041.751,415.341,363.711,174.602,44.693,158.940
C08198=1041.761,415.586,363.664,174.612,44.700,158.943
C08199=1041.772,415.832,363.618,174.623,44.707,158.946
C08200=1041.782,416.077,363.571,174.634,44.714,158.949
C08201=1041.792,416.322,363.524,174.644,44.721,158.952
C08202=1041.803,416.568,363.476,174.655,44.728,158.955
C08203=1041.814,416.813,363.430,174.666,44.734,158.958
C08204=1041.824,417.059,363.382,174.677,44.741,158.960
C08205=1041.835,417.304,363.335,174.687,44.748,158.963
C08206=1041.845,417.549,363.288,174.698,44.755,158.966
C08207=1041.856,417.794,363.241,174.709,44.762,158.969
C08208=1041.866,418.039,363.194,174.720,44.769,158.972
C08209=1041.877,418.285,363.146,174.730,44.776,158.975
C08210=1041.887,418.531,363.099,174.742,44.783,158.978
C08211=1041.897,418.775,363.051,174.753,44.791,158.981
C08212=1041.908,419.021,363.004,174.764,44.798,158.984
C08213=1041.918,419.267,362.956,174.775,44.805,158.987
C08214=1041.929,419.511,362.908,174.786,44.812,158.990
C08215=1041.939,419.756,362.861,174.797,44.819,158.993
C08216=1041.948,419.978,362.818,174.807,44.826,158.996
C08217=1041.958,420.199,362.775,174.818,44.832,158.999
C08218=1041.968,420.419,362.732,174.828,44.839,159.002
C08219=1041.977,420.640,362.688,174.838,44.846,159.005
C08220=1041.987,420.861,362.645,174.848,44.852,159.007
C08221=1041.997,421.082,362.602,174.858,44.858,159.010
C08222=1042.005,421.302,362.558,174.869,44.865,159.013
C08223=1042.015,421.523,362.516,174.879,44.871,159.016
C08224=1042.026,421.769,362.467,174.890,44.879,159.019
C08225=1042.037,422.013,362.419,174.902,44.886,159.022
C08226=1042.048,422.259,362.372,174.914,44.894,159.025
C08227=1042.058,422.504,362.324,174.925,44.902,159.028
C08228=1042.069,422.749,362.276,174.936,44.909,159.032
C08229=1042.081,422.994,362.227,174.949,44.916,159.035
C08230=1042.091,423.239,362.179,174.960,44.924,159.038
C08231=1042.102,423.484,362.130,174.972,44.931,159.041
C08232=1042.113,423.730,362.082,174.984,44.939,159.044
C08233=1042.124,423.975,362.033,174.996,44.946,159.048
C08234=1042.134,424.220,361.985,175.007,44.954,159.051
C08235=1042.146,424.465,361.936,175.020,44.962,159.054
C08236=1042.157,424.710,361.888,175.031,44.969,159.058
C08237=1042.168,424.955,361.839,175.044,44.977,159.061
C08238=1042.178,425.200,361.790,175.055,44.985,159.064
C08239=1042.189,425.444,361.741,175.068,44.992,159.068
C08240=1042.200,425.690,361.693,175.079,45.000,159.071
C08241=1042.211,425.935,361.643,175.092,45.008,159.074
C08242=1042.223,426.180,361.594,175.103,45.015,159.078
C08243=1042.234,426.424,361.545,175.116,45.024,159.081
C08244=1042.244,426.670,361.497,175.128,45.031,159.085
C08245=1042.256,426.915,361.447,175.141,45.039,159.088
C08246=1042.267,427.159,361.398,175.153,45.047,159.091
C08247=1042.279,427.404,361.349,175.165,45.055,159.095
C08248=1042.289,427.649,361.300,175.178,45.063,159.098
C08249=1042.301,427.894,361.251,175.191,45.071,159.102
C08250=1042.312,428.139,361.202,175.202,45.079,159.105
C08251=1042.323,428.384,361.152,175.215,45.087,159.109
C08252=1042.334,428.628,361.102,175.228,45.095,159.112
C08253=1042.346,428.874,361.053,175.241,45.103,159.116
C08254=1042.357,429.118,361.004,175.253,45.111,159.119
C08255=1042.368,429.363,360.953,175.266,45.119,159.123
C08256=1042.379,429.608,360.904,175.279,45.127,159.127
C08257=1042.390,429.852,360.854,175.292,45.136,159.130
C08258=1042.402,430.097,360.804,175.305,45.144,159.134
C08259=1042.413,430.342,360.754,175.318,45.152,159.137
C08260=1042.424,430.587,360.705,175.331,45.160,159.141
C08261=1042.436,430.832,360.654,175.344,45.168,159.145
C08262=1042.447,431.076,360.604,175.357,45.177,159.148
C08263=1042.459,431.320,360.554,175.370,45.185,159.152
C08264=1042.471,431.565,360.504,175.383,45.193,159.156
C08265=1042.482,431.810,360.454,175.396,45.202,159.160
C08266=1042.494,432.055,360.404,175.409,45.210,159.163
C08267=1042.505,432.300,360.354,175.423,45.219,159.167
C08268=1042.517,432.544,360.303,175.436,45.227,159.171
C08269=1042.528,432.788,360.253,175.450,45.236,159.175
C08270=1042.540,433.033,360.202,175.463,45.244,159.178
C08271=1042.551,433.278,360.152,175.476,45.253,159.182
C08272=1042.564,433.522,360.102,175.490,45.262,159.186
C08273=1042.576,433.767,360.051,175.504,45.270,159.190
C08274=1042.587,434.011,360.000,175.517,45.278,159.194
C08275=1042.599,434.256,359.950,175.531,45.287,159.198
C08276=1042.618,434.657,359.867,175.554,45.301,159.204
C08277=1042.638,435.057,359.783,175.576,45.315,159.210
C08278=1042.657,435.458,359.700,175.599,45.330,159.217
C08279=1042.677,435.857,359.617,175.622,45.344,159.223
C08280=1042.689,436.102,359.565,175.636,45.353,159.227
C08281=1042.701,436.346,359.514,175.651,45.362,159.231
C08282=1042.713,436.591,359.462,175.664,45.371,159.235
C08283=1042.726,436.835,359.412,175.679,45.380,159.239
C08284=1042.740,437.139,359.348,175.697,45.391,159.244
C08285=1042.755,437.442,359.284,175.714,45.402,159.250
C08286=1042.770,437.746,359.221,175.732,45.413,159.255
C08287=1042.785,438.048,359.156,175.750,45.424,159.260
C08288=1042.797,438.293,359.105,175.765,45.434,159.264
C08289=1042.809,438.537,359.052,175.780,45.443,159.268
C08290=1042.821,438.781,359.001,175.794,45.451,159.272
C08291=1042.834,439.025,358.949,175.808,45.461,159.276
C08292=1042.846,439.270,358.897,175.823,45.470,159.281
C08293=1042.859,439.514,358.846,175.838,45.480,159.285
C08294=1042.871,439.758,358.793,175.853,45.489,159.289
C08295=1042.884,440.003,358.742,175.868,45.498,159.294
C08296=1042.896,440.247,358.690,175.883,45.507,159.298
C08297=1042.908,440.491,358.637,175.898,45.517,159.302
C08298=1042.921,440.735,358.585,175.913,45.526,159.307
C08299=1042.933,440.979,358.533,175.929,45.535,159.311
C08300=1042.946,441.224,358.480,175.944,45.545,159.315
C08301=1042.958,441.468,358.428,175.960,45.554,159.320
C08302=1042.971,441.712,358.375,175.975,45.564,159.324
C08303=1042.983,441.956,358.323,175.990,45.573,159.329
C08304=1042.996,442.200,358.270,176.006,45.583,159.333
C08305=1043.008,442.444,358.218,176.021,45.592,159.337
C08306=1043.021,442.688,358.165,176.037,45.602,159.342
C08307=1043.034,442.932,358.111,176.053,45.611,159.346
C08308=1043.046,443.176,358.059,176.068,45.621,159.351
C08309=1043.059,443.420,358.006,176.084,45.631,159.355
C08310=1043.072,443.664,357.953,176.100,45.641,159.360
C08311=1043.085,443.909,357.900,176.116,45.651,159.365
C08312=1043.098,444.153,357.847,176.132,45.660,159.369
C08313=1043.110,444.396,357.794,176.148,45.670,159.374
C08314=1043.123,444.640,357.741,176.164,45.680,159.379
C08315=1043.137,444.884,357.688,176.181,45.689,159.383
C08316=1043.150,445.126,357.635,176.196,45.699,159.388
C08317=1043.163,445.369,357.583,176.213,45.709,159.393
C08318=1043.178,445.613,357.531,176.229,45.719,159.397
C08319=1043.193,445.857,357.479,176.245,45.728,159.402
C08320=1043.208,446.100,357.428,176.262,45.738,159.406
C08321=1043.224,446.344,357.377,176.278,45.747,159.411
C08322=1043.241,446.588,357.327,176.296,45.756,159.415
C08323=1043.259,446.832,357.277,176.312,45.765,159.420
C08324=1043.277,447.076,357.228,176.329,45.774,159.424
C08325=1043.295,447.320,357.179,176.346,45.783,159.429
C08326=1043.314,447.564,357.131,176.363,45.792,159.434
C08327=1043.334,447.809,357.083,176.380,45.800,159.438
C08328=1043.354,448.053,357.036,176.397,45.809,159.442
C08329=1043.375,448.298,356.989,176.415,45.817,159.447
C08330=1043.397,448.543,356.943,176.432,45.825,159.451
C08331=1043.420,448.787,356.896,176.449,45.833,159.455
C08332=1043.455,449.168,356.826,176.476,45.846,159.462
C08333=1043.492,449.549,356.757,176.503,45.858,159.469
C08334=1043.531,449.930,356.689,176.532,45.870,159.476
C08335=1043.571,450.311,356.623,176.559,45.881,159.482
C08336=1043.598,450.556,356.580,176.577,45.889,159.487
C08337=1043.625,450.802,356.539,176.595,45.897,159.491
C08338=1043.653,451.048,356.497,176.614,45.904,159.495
C08339=1043.681,451.292,356.457,176.631,45.910,159.499
C08340=1043.379,451.334,356.143,176.634,45.991,159.524
C08341=1043.351,451.089,356.184,176.616,45.984,159.519
C08342=1043.323,450.844,356.225,176.597,45.977,159.515
C08343=1043.295,450.598,356.267,176.579,45.970,159.511
C08344=1043.269,450.353,356.310,176.561,45.962,159.507
C08345=1043.230,449.987,356.373,176.535,45.951,159.500
C08346=1043.192,449.622,356.438,176.508,45.940,159.494
C08347=1043.157,449.257,356.504,176.481,45.929,159.488
C08348=1043.121,448.892,356.571,176.455,45.917,159.481
C08349=1043.099,448.648,356.617,176.437,45.909,159.477
C08350=1043.077,448.403,356.663,176.420,45.901,159.472
C08351=1043.056,448.158,356.709,176.403,45.893,159.468
C08352=1043.035,447.914,356.756,176.385,45.884,159.463
C08353=1043.015,447.669,356.804,176.368,45.876,159.459
C08354=1042.995,447.425,356.852,176.351,45.867,159.454
C08355=1042.976,447.180,356.900,176.335,45.859,159.450
C08356=1042.958,446.937,356.949,176.317,45.850,159.446
C08357=1042.940,446.692,356.999,176.300,45.841,159.441
C08358=1042.923,446.448,357.049,176.284,45.832,159.436
C08359=1042.907,446.204,357.099,176.267,45.823,159.432
C08360=1042.891,445.962,357.150,176.250,45.814,159.427
C08361=1042.875,445.717,357.201,176.233,45.804,159.423
C08362=1042.861,445.474,357.253,176.217,45.795,159.418
C08363=1042.847,445.230,357.306,176.201,45.785,159.413
C08364=1042.833,444.988,357.359,176.185,45.775,159.409
C08365=1042.820,444.744,357.412,176.168,45.765,159.404
C08366=1042.808,444.501,357.465,176.152,45.756,159.399
C08367=1042.795,444.257,357.518,176.136,45.746,159.395
C08368=1042.781,444.013,357.571,176.120,45.736,159.390
C08369=1042.769,443.768,357.623,176.103,45.727,159.386
C08370=1042.756,443.524,357.677,176.088,45.717,159.381
C08371=1042.743,443.281,357.730,176.072,45.707,159.376
C08372=1042.730,443.037,357.783,176.056,45.698,159.372
C08373=1042.717,442.792,357.835,176.040,45.689,159.367
C08374=1042.704,442.548,357.888,176.025,45.679,159.363
C08375=1042.692,442.305,357.941,176.009,45.669,159.358
C08376=1042.679,442.061,357.994,175.993,45.660,159.354
C08377=1042.667,441.817,358.046,175.978,45.651,159.350
C08378=1042.654,441.572,358.098,175.963,45.641,159.345
C08379=1042.642,441.328,358.150,175.947,45.631,159.341
C08380=1042.629,441.084,358.204,175.931,45.622,159.336
C08381=1042.616,440.840,358.256,175.916,45.613,159.332
C08382=1042.604,440.596,358.308,175.901,45.603,159.327
C08383=1042.591,440.352,358.360,175.886,45.594,159.323
C08384=1042.579,440.107,358.413,175.871,45.585,159.319
C08385=1042.567,439.863,358.464,175.856,45.576,159.315
C08386=1042.554,439.619,358.516,175.841,45.566,159.310
C08387=1042.542,439.374,358.569,175.826,45.557,159.306
C08388=1042.530,439.130,358.621,175.811,45.548,159.302
C08389=1042.517,438.886,358.672,175.796,45.539,159.298
C08390=1042.504,438.642,358.724,175.781,45.530,159.293
C08391=1042.492,438.397,358.776,175.767,45.521,159.289
C08392=1042.480,438.153,358.828,175.752,45.512,159.285
C08393=1042.468,437.909,358.879,175.737,45.503,159.281
C08394=1042.456,437.665,358.931,175.723,45.494,159.277
C08395=1042.444,437.420,358.983,175.709,45.485,159.273
C08396=1042.432,437.176,359.034,175.694,45.476,159.269
C08397=1042.420,436.932,359.085,175.679,45.467,159.264
C08398=1042.408,436.687,359.136,175.666,45.458,159.260
C08399=1042.396,436.443,359.188,175.651,45.450,159.256
C08400=1042.384,436.198,359.239,175.636,45.441,159.252
C08401=1042.372,435.968,359.288,175.623,45.433,159.249
C08402=1042.361,435.737,359.336,175.610,45.424,159.245
C08403=1042.350,435.507,359.383,175.596,45.416,159.241
C08404=1042.338,435.277,359.432,175.583,45.408,159.237
C08405=1042.327,435.046,359.480,175.570,45.400,159.234
C08406=1042.316,434.815,359.528,175.557,45.392,159.230
C08407=1042.305,434.585,359.576,175.544,45.383,159.226
C08408=1042.294,434.355,359.624,175.531,45.376,159.223
C08409=1042.281,434.110,359.674,175.517,45.367,159.219
C08410=1042.270,433.865,359.725,175.503,45.358,159.215
C08411=1042.257,433.621,359.775,175.490,45.350,159.211
C08412=1042.246,433.377,359.826,175.477,45.341,159.207
C08413=1042.234,433.132,359.876,175.463,45.332,159.203
C08414=1042.223,432.887,359.927,175.449,45.324,159.199
C08415=1042.211,432.642,359.977,175.436,45.316,159.196
C08416=1042.199,432.397,360.027,175.422,45.307,159.192
C08417=1042.188,432.153,360.078,175.409,45.299,159.188
C08418=1042.176,431.908,360.128,175.395,45.291,159.184
C08419=1042.165,431.664,360.178,175.382,45.283,159.181
C08420=1042.152,431.419,360.228,175.369,45.274,159.177
C08421=1042.133,431.022,360.310,175.348,45.261,159.171
C08422=1042.115,430.624,360.391,175.326,45.248,159.165
C08423=1042.097,430.226,360.472,175.305,45.234,159.159
C08424=1042.079,429.829,360.553,175.284,45.221,159.153
C08425=1042.066,429.584,360.603,175.271,45.213,159.150
C08426=1042.056,429.339,360.653,175.258,45.205,159.146
C08427=1042.045,429.094,360.703,175.245,45.197,159.142
C08428=1042.033,428.850,360.752,175.233,45.189,159.139
C08429=1042.022,428.605,360.802,175.220,45.181,159.135
C08430=1042.010,428.360,360.852,175.207,45.173,159.132
C08431=1042.000,428.115,360.901,175.194,45.165,159.128
C08432=1041.988,427.870,360.950,175.182,45.157,159.125
C08433=1041.977,427.625,360.999,175.170,45.149,159.121
C08434=1041.966,427.380,361.048,175.157,45.141,159.118
C08435=1041.955,427.135,361.098,175.144,45.133,159.114
C08436=1041.943,426.891,361.147,175.133,45.126,159.111
C08437=1041.932,426.646,361.196,175.120,45.117,159.107
C08438=1041.921,426.401,361.246,175.107,45.110,159.104
C08439=1041.910,426.156,361.295,175.096,45.102,159.101
C08440=1041.899,425.911,361.343,175.083,45.094,159.097
C08441=1041.888,425.666,361.393,175.070,45.087,159.094
C08442=1041.877,425.421,361.442,175.059,45.079,159.091
C08443=1041.866,425.176,361.490,175.046,45.071,159.087
C08444=1041.854,424.931,361.539,175.035,45.064,159.084
C08445=1041.845,424.686,361.587,175.022,45.056,159.081
C08446=1041.833,424.441,361.636,175.010,45.048,159.077
C08447=1041.822,424.196,361.685,174.999,45.041,159.074
C08448=1041.811,423.950,361.733,174.987,45.033,159.071
C08449=1041.800,423.706,361.782,174.975,45.026,159.067
C08450=1041.789,423.461,361.830,174.963,45.019,159.064
C08451=1041.778,423.216,361.878,174.951,45.011,159.061
C08452=1041.767,422.970,361.927,174.940,45.004,159.058
C08453=1041.756,422.726,361.974,174.927,44.996,159.054
C08454=1041.746,422.480,362.023,174.916,44.989,159.051
C08455=1041.735,422.235,362.072,174.905,44.981,159.048
C08456=1041.724,421.990,362.120,174.892,44.974,159.045
C08457=1041.713,421.745,362.168,174.881,44.967,159.042
C08458=1041.703,421.500,362.216,174.870,44.959,159.039
C08459=1041.692,421.255,362.264,174.858,44.952,159.035
C08460=1041.681,421.010,362.312,174.847,44.945,159.032
C08461=1041.668,420.719,362.369,174.833,44.936,159.029
C08462=1041.655,420.428,362.425,174.820,44.927,159.025
C08463=1041.643,420.138,362.482,174.806,44.919,159.021
C08464=1041.631,419.847,362.539,174.793,44.911,159.018
C08465=1041.620,419.601,362.586,174.782,44.903,159.015
C08466=1041.610,419.356,362.634,174.771,44.896,159.011
C08467=1041.599,419.111,362.682,174.760,44.889,159.009
C08468=1041.589,418.866,362.730,174.748,44.882,159.005
C08469=1041.578,418.620,362.777,174.737,44.875,159.003
C08470=1041.568,418.375,362.824,174.726,44.868,158.999
C08471=1041.558,418.130,362.872,174.715,44.861,158.996
C08472=1041.547,417.885,362.919,174.704,44.854,158.994
C08473=1041.536,417.639,362.966,174.693,44.847,158.990
C08474=1041.526,417.394,363.014,174.682,44.840,158.988
C08475=1041.515,417.149,363.061,174.671,44.833,158.985
C08476=1041.505,416.904,363.108,174.660,44.826,158.982
C08477=1041.494,416.659,363.155,174.650,44.819,158.979
C08478=1041.484,416.413,363.202,174.639,44.813,158.976
C08479=1041.473,416.167,363.250,174.628,44.806,158.973
C08480=1041.463,415.921,363.296,174.617,44.799,158.970
C08481=1041.452,415.676,363.343,174.606,44.792,158.967
C08482=1041.442,415.431,363.390,174.597,44.786,158.964
C08483=1041.432,415.186,363.437,174.586,44.779,158.962
C08484=1041.422,414.940,363.484,174.575,44.772,158.959
C08485=1041.411,414.695,363.530,174.564,44.766,158.956
C08486=1041.401,414.450,363.577,174.554,44.759,158.953
C08487=1041.392,414.205,363.624,174.543,44.752,158.950
C08488=1041.382,413.959,363.671,174.534,44.745,158.947
C08489=1041.371,413.714,363.717,174.523,44.738,158.945
C08490=1041.361,413.468,363.764,174.512,44.732,158.942
C08491=1041.351,413.222,363.810,174.502,44.725,158.939
C08492=1041.340,412.977,363.856,174.491,44.719,158.936
C08493=1041.331,412.732,363.903,174.482,44.712,158.934
C08494=1041.321,412.486,363.950,174.471,44.706,158.931
C08495=1041.311,412.241,363.996,174.460,44.699,158.928
C08496=1041.300,411.995,364.042,174.451,44.693,158.925
C08497=1041.291,411.750,364.088,174.440,44.687,158.923
C08498=1041.280,411.504,364.134,174.430,44.680,158.920
C08499=1041.271,411.258,364.181,174.420,44.674,158.917
C08500=1041.260,411.013,364.227,174.410,44.667,158.915
C08501=1041.251,410.767,364.273,174.401,44.661,158.912
C08502=1041.240,410.522,364.319,174.390,44.654,158.909
C08503=1041.229,410.276,364.364,174.381,44.648,158.907
C08504=1041.220,410.030,364.410,174.370,44.642,158.904
C08505=1041.210,409.785,364.456,174.360,44.635,158.901
C08506=1041.201,409.540,364.502,174.351,44.629,158.899
C08507=1041.190,409.294,364.548,174.340,44.623,158.896
C08508=1041.180,409.048,364.593,174.331,44.617,158.894
C08509=1041.170,408.803,364.639,174.321,44.610,158.891
C08510=1041.161,408.557,364.684,174.311,44.604,158.888
C08511=1041.151,408.311,364.730,174.301,44.598,158.886
C08512=1041.141,408.066,364.775,174.292,44.592,158.883
C08513=1041.130,407.820,364.821,174.282,44.586,158.881
C08514=1041.121,407.574,364.867,174.272,44.580,158.878
C08515=1041.111,407.329,364.912,174.263,44.573,158.876
C08516=1041.101,407.083,364.957,174.253,44.567,158.873
C08517=1041.093,406.865,364.998,174.245,44.562,158.871
C08518=1041.084,406.647,365.038,174.236,44.557,158.869
C08519=1041.075,406.429,365.078,174.227,44.551,158.866
C08520=1041.067,406.211,365.119,174.220,44.546,158.864
C08521=1041.058,405.993,365.158,174.210,44.540,158.862
C08522=1041.050,405.776,365.198,174.203,44.535,158.860
C08523=1041.042,405.558,365.239,174.195,44.530,158.858
C08524=1041.033,405.340,365.278,174.186,44.525,158.856
C08525=1041.023,405.095,365.323,174.176,44.519,158.853
C08526=1041.014,404.848,365.369,174.167,44.513,158.851
C08527=1041.004,404.603,365.414,174.158,44.507,158.848
C08528=1040.994,404.357,365.459,174.149,44.501,158.846
C08529=1040.985,404.111,365.504,174.139,44.495,158.843
C08530=1040.976,403.866,365.549,174.130,44.489,158.841
C08531=1040.966,403.620,365.594,174.121,44.483,158.839
C08532=1040.957,403.375,365.639,174.112,44.477,158.836
C08533=1040.947,403.128,365.683,174.103,44.472,158.834
C08534=1040.938,402.883,365.728,174.094,44.466,158.831
C08535=1040.928,402.637,365.773,174.084,44.460,158.829
C08536=1040.919,402.391,365.817,174.075,44.454,158.827
C08537=1040.909,402.146,365.862,174.066,44.448,158.824
C08538=1040.900,401.899,365.907,174.057,44.443,158.822
C08539=1040.891,401.654,365.951,174.048,44.437,158.820
C08540=1040.881,401.408,365.995,174.039,44.432,158.817
C08541=1040.871,401.162,366.040,174.030,44.426,158.815
C08542=1040.862,400.916,366.084,174.021,44.421,158.813
C08543=1040.853,400.671,366.129,174.012,44.414,158.810
C08544=1040.843,400.425,366.173,174.003,44.409,158.808
C08545=1040.834,400.179,366.217,173.994,44.403,158.806
C08546=1040.825,399.933,366.261,173.985,44.398,158.804
C08547=1040.815,399.687,366.306,173.976,44.393,158.801
C08548=1040.806,399.442,366.350,173.967,44.387,158.799
C08549=1040.797,399.196,366.394,173.959,44.381,158.797
C08550=1040.787,398.950,366.438,173.950,44.376,158.795
C08551=1040.778,398.703,366.482,173.941,44.371,158.792
C08552=1040.768,398.458,366.525,173.932,44.365,158.790
C08553=1040.759,398.212,366.569,173.924,44.359,158.788
C08554=1040.750,397.966,366.613,173.916,44.354,158.786
C08555=1040.741,397.721,366.657,173.907,44.349,158.784
C08556=1040.731,397.474,366.701,173.898,44.343,158.781
C08557=1040.722,397.229,366.745,173.890,44.338,158.779
C08558=1040.713,396.983,366.789,173.881,44.332,158.777
C08559=1040.704,396.736,366.833,173.872,44.327,158.775
C08560=1040.694,396.491,366.876,173.864,44.321,158.773
C08561=1040.685,396.245,366.920,173.855,44.316,158.770
C08562=1040.676,395.999,366.964,173.847,44.311,158.768
C08563=1040.667,395.753,367.007,173.838,44.305,158.766
C08564=1040.658,395.507,367.051,173.830,44.300,158.764
C08565=1040.649,395.261,367.095,173.822,44.295,158.762
C08566=1040.640,395.015,367.137,173.813,44.290,158.760
C08567=1040.630,394.769,367.181,173.804,44.285,158.758
C08568=1040.622,394.523,367.224,173.797,44.280,158.756
C08569=1040.613,394.277,367.267,173.788,44.274,158.753
C08570=1040.603,394.031,367.311,173.780,44.269,158.751
C08571=1040.595,393.785,367.354,173.771,44.264,158.749
C08572=1040.584,393.539,367.397,173.763,44.259,158.747
C08573=1040.576,393.293,367.440,173.755,44.254,158.745
C08574=1040.567,393.047,367.484,173.747,44.249,158.743
C08575=1040.558,392.801,367.527,173.738,44.244,158.741
C08576=1040.549,392.555,367.570,173.731,44.238,158.739
C08577=1040.534,392.139,367.643,173.716,44.230,158.736
C08578=1040.519,391.723,367.716,173.703,44.222,158.732
C08579=1040.504,391.306,367.788,173.689,44.213,158.729
C08580=1040.489,390.891,367.860,173.676,44.205,158.725
C08581=1040.479,390.644,367.903,173.667,44.200,158.723
C08582=1040.471,390.398,367.946,173.659,44.194,158.721
C08583=1040.462,390.152,367.988,173.652,44.190,158.719
C08584=1040.453,389.906,368.031,173.643,44.185,158.718
C08585=1040.444,389.661,368.074,173.636,44.180,158.716
C08586=1040.436,389.414,368.116,173.627,44.175,158.714
C08587=1040.426,389.168,368.158,173.619,44.170,158.712
C08588=1040.417,388.921,368.202,173.612,44.165,158.710
C08589=1040.408,388.676,368.244,173.603,44.161,158.708
C08590=1040.400,388.429,368.286,173.596,44.155,158.706
C08591=1040.391,388.183,368.329,173.588,44.151,158.704
C08592=1040.382,387.937,368.371,173.581,44.146,158.702
C08593=1040.373,387.691,368.414,173.572,44.141,158.700
C08594=1040.364,387.444,368.455,173.565,44.137,158.698
C08595=1040.356,387.198,368.498,173.557,44.132,158.696
C08596=1040.347,386.952,368.540,173.549,44.127,158.694
C08597=1040.338,386.706,368.582,173.541,44.123,158.693
C08598=1040.329,386.460,368.624,173.534,44.118,158.691
C08599=1040.320,386.213,368.667,173.527,44.113,158.689
C08600=1040.312,385.967,368.708,173.518,44.109,158.687
C08601=1040.303,385.720,368.750,173.511,44.104,158.685
C08602=1040.293,385.475,368.792,173.503,44.099,158.683
C08603=1040.285,385.229,368.834,173.496,44.095,158.681
C08604=1040.277,384.982,368.876,173.489,44.090,158.680
C08605=1040.268,384.736,368.918,173.480,44.085,158.678
C08606=1040.259,384.490,368.960,173.473,44.081,158.676
C08607=1040.250,384.243,369.001,173.465,44.077,158.674
C08608=1040.242,383.997,369.044,173.458,44.072,158.672
C08609=1040.233,383.751,369.085,173.450,44.067,158.670
C08610=1040.225,383.505,369.127,173.443,44.063,158.669
C08611=1040.216,383.258,369.168,173.436,44.058,158.667
C08612=1040.207,383.012,369.210,173.429,44.054,158.665
C08613=1040.198,382.765,369.252,173.420,44.049,158.663
C08614=1040.190,382.520,369.294,173.413,44.045,158.662
C08615=1040.181,382.273,369.335,173.406,44.040,158.660
C08616=1040.172,382.027,369.377,173.398,44.036,158.658
C08617=1040.164,381.781,369.418,173.391,44.031,158.656
C08618=1040.156,381.534,369.460,173.384,44.027,158.654
C08619=1040.147,381.287,369.502,173.376,44.022,158.653
C08620=1040.139,381.041,369.542,173.369,44.018,158.651
C08621=1040.130,380.795,369.584,173.362,44.014,158.649
C08622=1040.122,380.549,369.626,173.355,44.010,158.648
C08623=1040.114,380.302,369.667,173.347,44.005,158.646
C08624=1040.106,380.056,369.708,173.340,44.001,158.644
C08625=1040.097,379.810,369.750,173.333,43.996,158.642
C08626=1040.088,379.563,369.791,173.326,43.992,158.641
C08627=1040.080,379.317,369.833,173.318,43.987,158.639
C08628=1040.071,379.070,369.874,173.311,43.983,158.637
C08629=1040.064,378.824,369.915,173.304,43.979,158.635
C08630=1040.055,378.577,369.956,173.297,43.975,158.634
C08631=1040.046,378.331,369.997,173.289,43.970,158.632
C08632=1040.037,378.084,370.038,173.283,43.966,158.630
C08633=1040.025,377.702,370.101,173.272,43.959,158.628
C08634=1040.012,377.320,370.165,173.261,43.953,158.625
C08635=1039.998,376.938,370.228,173.250,43.947,158.623
C08636=1039.985,376.556,370.292,173.239,43.941,158.620
C08637=1039.977,376.310,370.332,173.232,43.936,158.619
C08638=1039.968,376.063,370.373,173.225,43.932,158.617
C08639=1039.960,375.817,370.413,173.219,43.928,158.615
C08640=1039.952,375.571,370.454,173.212,43.924,158.614
C08641=1039.943,375.324,370.495,173.205,43.920,158.612
C08642=1039.935,375.077,370.536,173.197,43.916,158.610
C08643=1039.927,374.831,370.575,173.190,43.912,158.609
C08644=1039.918,374.584,370.616,173.183,43.908,158.607
C08645=1039.910,374.338,370.656,173.177,43.904,158.606
C08646=1039.902,374.091,370.697,173.170,43.900,158.604
C08647=1039.894,373.845,370.738,173.163,43.896,158.602
C08648=1039.885,373.598,370.779,173.156,43.892,158.601
C08649=1039.878,373.351,370.819,173.150,43.888,158.599
C08650=1039.869,373.105,370.859,173.143,43.883,158.598
C08651=1039.861,372.859,370.899,173.136,43.880,158.596
C08652=1039.853,372.612,370.939,173.129,43.875,158.594
C08653=1039.845,372.365,370.980,173.123,43.872,158.593
C08654=1039.837,372.119,371.021,173.116,43.868,158.592
C08655=1039.828,371.872,371.060,173.109,43.864,158.590
C08656=1039.820,371.626,371.101,173.102,43.860,158.588
C08657=1039.812,371.379,371.141,173.096,43.856,158.587
C08658=1039.804,371.133,371.181,173.089,43.852,158.585
C08659=1039.797,370.886,371.221,173.082,43.848,158.584
C08660=1039.788,370.640,371.261,173.076,43.844,158.582
C08661=1039.779,370.392,371.302,173.069,43.840,158.581
C08662=1039.771,370.146,371.342,173.062,43.837,158.579
C08663=1039.763,369.899,371.382,173.056,43.833,158.578
C08664=1039.755,369.652,371.422,173.049,43.829,158.576
C08665=1039.747,369.406,371.461,173.042,43.825,158.575
C08666=1039.739,369.160,371.501,173.037,43.822,158.573
C08667=1039.730,368.913,371.541,173.030,43.818,158.572
C08668=1039.723,368.666,371.581,173.024,43.814,158.570
C08669=1039.714,368.419,371.620,173.017,43.810,158.569
C08670=1039.706,368.172,371.660,173.010,43.807,158.567
C08671=1039.698,367.926,371.699,173.004,43.803,158.566
C08672=1039.690,367.679,371.739,172.997,43.799,158.564
C08673=1039.682,367.432,371.779,172.991,43.796,158.563
C08674=1039.674,367.185,371.818,172.985,43.792,158.562
C08675=1039.666,366.939,371.858,172.978,43.788,158.560
C08676=1039.657,366.692,371.897,172.972,43.784,158.559
C08677=1039.649,366.445,371.937,172.965,43.781,158.557
C08678=1039.641,366.199,371.976,172.959,43.777,158.556
C08679=1039.633,365.952,372.016,172.952,43.773,158.554
C08680=1039.625,365.705,372.056,172.947,43.770,158.553
C08681=1039.618,365.459,372.095,172.940,43.766,158.551
C08682=1039.609,365.213,372.134,172.934,43.763,158.550
C08683=1039.602,364.965,372.174,172.927,43.759,158.549
C08684=1039.593,364.718,372.213,172.921,43.755,158.547
C08685=1039.586,364.471,372.253,172.914,43.752,158.546
C08686=1039.578,364.226,372.292,172.909,43.748,158.544
C08687=1039.570,363.978,372.330,172.902,43.745,158.543
C08688=1039.562,363.731,372.370,172.896,43.741,158.542
C08689=1039.550,363.370,372.428,172.886,43.736,158.540
C08690=1039.539,363.008,372.485,172.878,43.731,158.538
C08691=1039.527,362.646,372.543,172.868,43.726,158.536
C08692=1039.516,362.283,372.601,172.860,43.720,158.534
C08693=1039.508,362.037,372.639,172.853,43.717,158.532
C08694=1039.500,361.790,372.679,172.847,43.713,158.531
C08695=1039.492,361.542,372.717,172.840,43.710,158.529
C08696=1039.484,361.297,372.756,172.835,43.707,158.528
C08697=1039.476,361.049,372.795,172.829,43.703,158.527
C08698=1039.468,360.802,372.833,172.822,43.700,158.525
C08699=1039.461,360.556,372.873,172.817,43.696,158.524
C08700=1039.453,360.309,372.912,172.810,43.693,158.523
C08701=1039.445,360.061,372.950,172.804,43.690,158.521
C08702=1039.437,359.815,372.988,172.799,43.686,158.520
C08703=1039.429,359.568,373.027,172.792,43.683,158.519
C08704=1039.420,359.321,373.066,172.786,43.680,158.518
C08705=1039.413,359.075,373.105,172.781,43.677,158.516
C08706=1039.405,358.827,373.143,172.774,43.673,158.515
C08707=1039.398,358.581,373.182,172.768,43.670,158.514
C08708=1039.390,358.333,373.221,172.763,43.667,158.512
C08709=1039.382,358.087,373.259,172.756,43.664,158.511
C08710=1039.374,357.840,373.298,172.750,43.660,158.510
C08711=1039.367,357.593,373.336,172.745,43.657,158.508
C08712=1039.358,357.346,373.374,172.738,43.654,158.507
C08713=1039.351,357.099,373.413,172.732,43.650,158.506
C08714=1039.343,356.852,373.451,172.727,43.647,158.505
C08715=1039.335,356.606,373.490,172.721,43.643,158.503
C08716=1039.328,356.358,373.529,172.715,43.640,158.502
C08717=1039.319,356.112,373.566,172.709,43.638,158.501
C08718=1039.312,355.864,373.604,172.703,43.634,158.500
C08719=1039.304,355.618,373.642,172.698,43.631,158.498
C08720=1039.296,355.370,373.681,172.691,43.628,158.497
C08721=1039.288,355.124,373.719,172.686,43.625,158.496
C08722=1039.281,354.877,373.757,172.680,43.621,158.495
C08723=1039.273,354.630,373.795,172.674,43.618,158.493
C08724=1039.265,354.383,373.834,172.668,43.615,158.492
C08725=1039.258,354.135,373.872,172.662,43.612,158.491
C08726=1039.250,353.889,373.910,172.657,43.609,158.490
C08727=1039.243,353.642,373.947,172.651,43.606,158.488
C08728=1039.234,353.395,373.985,172.645,43.603,158.487
C08729=1039.226,353.148,374.024,172.639,43.600,158.486
C08730=1039.219,352.901,374.061,172.634,43.597,158.485
C08731=1039.211,352.654,374.100,172.628,43.594,158.484
C08732=1039.204,352.407,374.137,172.623,43.590,158.482
C08733=1039.196,352.160,374.176,172.617,43.588,158.481
C08734=1039.189,351.913,374.213,172.611,43.584,158.480
C08735=1039.181,351.665,374.251,172.605,43.582,158.479
C08736=1039.174,351.419,374.289,172.600,43.578,158.477
C08737=1039.166,351.172,374.326,172.594,43.575,158.476
C08738=1039.158,350.925,374.364,172.589,43.572,158.475
C08739=1039.150,350.677,374.402,172.583,43.569,158.474
C08740=1039.143,350.430,374.440,172.578,43.566,158.473
C08741=1039.136,350.183,374.477,172.571,43.563,158.472
C08742=1039.128,349.937,374.516,172.566,43.560,158.470
C08743=1039.120,349.690,374.553,172.560,43.558,158.469
C08744=1039.113,349.443,374.590,172.555,43.554,158.468
C08745=1039.102,349.087,374.645,172.547,43.550,158.467
C08746=1039.091,348.730,374.698,172.539,43.546,158.465
C08747=1039.079,348.374,374.752,172.531,43.542,158.463
C08748=1039.069,348.018,374.806,172.524,43.538,158.462
C08749=1039.061,347.771,374.843,172.517,43.535,158.460
C08750=1039.054,347.524,374.881,172.512,43.532,158.459
C08751=1039.046,347.277,374.918,172.506,43.529,158.458
C08752=1039.038,347.030,374.955,172.501,43.526,158.457
C08753=1039.031,346.783,374.993,172.495,43.523,158.456
C08754=1039.023,346.536,375.030,172.490,43.520,158.455
C08755=1039.016,346.289,375.067,172.485,43.518,158.454
C08756=1039.009,346.041,375.105,172.479,43.515,158.452
C08757=1039.001,345.795,375.142,172.474,43.512,158.451
C08758=1038.993,345.547,375.179,172.468,43.509,158.450
C08759=1038.986,345.300,375.215,172.463,43.506,158.449
C08760=1038.979,345.053,375.253,172.458,43.503,158.448
C08761=1038.971,344.806,375.290,172.452,43.501,158.447
C08762=1038.963,344.559,375.327,172.447,43.498,158.446
C08763=1038.956,344.312,375.364,172.442,43.496,158.445
C08764=1038.948,344.064,375.401,172.436,43.493,158.444
C08765=1038.941,343.817,375.439,172.431,43.490,158.443
C08766=1038.933,343.570,375.475,172.425,43.487,158.442
C08767=1038.926,343.323,375.512,172.420,43.484,158.440
C08768=1038.919,343.075,375.549,172.415,43.481,158.439
C08769=1038.911,342.828,375.586,172.410,43.479,158.438
C08770=1038.903,342.581,375.623,172.404,43.476,158.437
C08771=1038.897,342.334,375.659,172.400,43.473,158.436
C08772=1038.889,342.087,375.696,172.394,43.470,158.435
C08773=1038.882,341.840,375.733,172.389,43.468,158.434
C08774=1038.874,341.593,375.770,172.384,43.465,158.433
C08775=1038.866,341.345,375.806,172.378,43.463,158.432
C08776=1038.859,341.098,375.843,172.373,43.460,158.431
C08777=1038.851,340.851,375.880,172.368,43.457,158.430
C08778=1038.844,340.604,375.916,172.363,43.455,158.429
C08779=1038.837,340.357,375.952,172.357,43.452,158.428
C08780=1038.829,340.109,375.990,172.352,43.450,158.427
C08781=1038.822,339.862,376.026,172.347,43.447,158.426
C08782=1038.814,339.615,376.062,172.341,43.444,158.425
C08783=1038.807,339.367,376.099,172.337,43.441,158.424
C08784=1038.800,339.121,376.136,172.332,43.439,158.423
C08785=1038.792,338.873,376.172,172.327,43.436,158.422
C08786=1038.784,338.626,376.208,172.321,43.434,158.421
C08787=1038.778,338.378,376.245,172.316,43.432,158.420
C08788=1038.770,338.131,376.281,172.311,43.429,158.419
C08789=1038.763,337.884,376.317,172.306,43.427,158.418
C08790=1038.755,337.637,376.354,172.301,43.424,158.417
C08791=1038.748,337.390,376.390,172.296,43.421,158.416
C08792=1038.741,337.143,376.426,172.291,43.419,158.414
C08793=1038.733,336.895,376.463,172.286,43.416,158.414
C08794=1038.726,336.648,376.498,172.280,43.414,158.413
C08795=1038.719,336.401,376.535,172.275,43.411,158.411
C08796=1038.711,336.153,376.572,172.271,43.409,158.411
C08797=1038.704,335.906,376.607,172.266,43.406,158.409
C08798=1038.697,335.659,376.644,172.260,43.404,158.409
C08799=1038.689,335.411,376.680,172.255,43.401,158.408
C08800=1038.683,335.164,376.716,172.250,43.399,158.407
C08801=1038.671,334.805,376.768,172.243,43.395,158.405
C08802=1038.661,334.445,376.820,172.235,43.392,158.404
C08803=1038.650,334.085,376.873,172.229,43.388,158.402
C08804=1038.639,333.726,376.925,172.221,43.385,158.401
C08805=1038.632,333.478,376.960,172.217,43.382,158.400
C08806=1038.625,333.231,376.996,172.212,43.380,158.399
C08807=1038.617,332.984,377.032,172.207,43.378,158.398
C08808=1038.610,332.736,377.068,172.201,43.375,158.397
C08809=1038.603,332.489,377.104,172.197,43.373,158.396
C08810=1038.595,332.242,377.140,172.192,43.371,158.395
C08811=1038.588,331.994,377.175,172.187,43.368,158.394
C08812=1038.581,331.747,377.211,172.182,43.366,158.393
C08813=1038.574,331.500,377.246,172.178,43.364,158.393
C08814=1038.566,331.252,377.282,172.173,43.361,158.392
C08815=1038.559,331.005,377.318,172.167,43.359,158.390
C08816=1038.552,330.757,377.354,172.163,43.356,158.390
C08817=1038.545,330.510,377.389,172.158,43.354,158.389
C08818=1038.538,330.263,377.425,172.153,43.352,158.388
C08819=1038.530,330.015,377.460,172.149,43.350,158.387
C08820=1038.523,329.768,377.496,172.144,43.348,158.386
C08821=1038.516,329.520,377.532,172.139,43.345,158.385
C08822=1038.509,329.274,377.568,172.133,43.343,158.384
C08823=1038.502,329.026,377.603,172.129,43.340,158.383
C08824=1038.495,328.778,377.638,172.124,43.338,158.382
C08825=1038.488,328.531,377.674,172.119,43.336,158.381
C08826=1038.480,328.284,377.709,172.115,43.333,158.380
C08827=1038.473,328.036,377.744,172.110,43.332,158.380
C08828=1038.465,327.789,377.779,172.105,43.330,158.379
C08829=1038.458,327.541,377.814,172.101,43.327,158.378
C08830=1038.450,327.295,377.849,172.096,43.325,158.377
C08831=1038.443,327.047,377.885,172.091,43.323,158.376
C08832=1038.435,326.800,377.919,172.086,43.321,158.375
C08833=1038.429,326.552,377.955,172.081,43.318,158.374
C08834=1038.421,326.304,377.990,172.076,43.317,158.374
C08835=1038.414,326.057,378.025,172.072,43.314,158.373
C08836=1038.406,325.809,378.060,172.067,43.312,158.372
C08837=1038.399,325.562,378.095,172.062,43.310,158.371
C08838=1038.392,325.315,378.130,172.058,43.308,158.370
C08839=1038.385,325.068,378.164,172.053,43.306,158.369
C08840=1038.377,324.820,378.200,172.049,43.304,158.368
C08841=1038.370,324.572,378.234,172.044,43.301,158.367
C08842=1038.363,324.325,378.269,172.039,43.300,158.367
C08843=1038.355,324.077,378.304,172.035,43.297,158.366
C08844=1038.348,323.830,378.340,172.030,43.296,158.365
C08845=1038.341,323.583,378.374,172.026,43.293,158.364
C08846=1038.334,323.335,378.408,172.021,43.291,158.363
C08847=1038.326,323.087,378.443,172.016,43.289,158.362
C08848=1038.319,322.840,378.479,172.012,43.287,158.362
C08849=1038.312,322.593,378.513,172.007,43.285,158.361
C08850=1038.305,322.345,378.548,172.003,43.283,158.360
C08851=1038.297,322.098,378.583,171.998,43.281,158.359
C08852=1038.291,321.850,378.617,171.994,43.279,158.358
C08853=1038.284,321.602,378.653,171.989,43.277,158.357
C08854=1038.276,321.355,378.687,171.984,43.275,158.357
C08855=1038.269,321.108,378.722,171.980,43.272,158.356
C08856=1038.262,320.860,378.756,171.975,43.271,158.355
C08857=1038.252,320.496,378.807,171.968,43.268,158.354
C08858=1038.241,320.132,378.858,171.962,43.265,158.352
C08859=1038.230,319.768,378.910,171.955,43.262,158.351
C08860=1038.220,319.404,378.960,171.949,43.259,158.350
C08861=1038.213,319.156,378.995,171.944,43.257,158.349
C08862=1038.206,318.909,379.029,171.940,43.255,158.348
C08863=1038.199,318.661,379.064,171.935,43.253,158.348
C08864=1038.192,318.413,379.098,171.931,43.251,158.347
C08865=1038.185,318.166,379.133,171.926,43.249,158.346
C08866=1038.178,317.918,379.167,171.922,43.247,158.345
C08867=1038.171,317.670,379.202,171.917,43.245,158.344
C08868=1038.164,317.423,379.236,171.913,43.243,158.344
C08869=1038.157,317.175,379.270,171.908,43.241,158.343
C08870=1038.150,316.928,379.305,171.904,43.239,158.342
C08871=1038.143,316.680,379.339,171.900,43.237,158.341
C08872=1038.136,316.433,379.374,171.895,43.235,158.340
C08873=1038.129,316.185,379.408,171.891,43.233,158.340
C08874=1038.122,315.938,379.442,171.886,43.231,158.339
C08875=1038.115,315.691,379.476,171.882,43.229,158.338
C08876=1038.109,315.443,379.511,171.877,43.228,158.337
C08877=1038.102,315.196,379.545,171.873,43.225,158.336
C08878=1038.095,314.948,379.580,171.869,43.223,158.336
C08879=1038.088,314.701,379.614,171.864,43.222,158.335
C08880=1038.081,314.453,379.648,171.861,43.220,158.334
C08881=1038.074,314.206,379.683,171.856,43.218,158.333
C08882=1038.067,313.958,379.716,171.852,43.215,158.332
C08883=1038.061,313.711,379.750,171.848,43.214,158.332
C08884=1038.053,313.463,379.784,171.843,43.212,158.331
C08885=1038.047,313.215,379.819,171.839,43.210,158.330
C08886=1038.039,312.968,379.853,171.834,43.208,158.329
C08887=1038.033,312.720,379.888,171.830,43.206,158.329
C08888=1038.026,312.473,379.921,171.826,43.205,158.328
C08889=1038.019,312.225,379.955,171.821,43.202,158.327
C08890=1038.013,311.977,379.989,171.817,43.200,158.326
C08891=1038.006,311.730,380.023,171.813,43.198,158.326
C08892=1037.999,311.483,380.057,171.808,43.197,158.325
C08893=1037.992,311.235,380.090,171.805,43.195,158.324
C08894=1037.984,310.988,380.124,171.800,43.194,158.323
C08895=1037.977,310.740,380.157,171.796,43.192,158.323
C08896=1037.969,310.492,380.191,171.792,43.190,158.322
C08897=1037.962,310.245,380.225,171.787,43.188,158.321
C08898=1037.955,309.996,380.258,171.783,43.187,158.321
C08899=1037.949,309.749,380.292,171.778,43.185,158.320
C08900=1037.941,309.502,380.325,171.774,43.183,158.319
C08901=1037.934,309.254,380.359,171.771,43.181,158.318
C08902=1037.926,309.007,380.393,171.766,43.180,158.318
C08903=1037.920,308.759,380.425,171.762,43.178,158.317
C08904=1037.913,308.511,380.459,171.758,43.177,158.316
C08905=1037.906,308.264,380.493,171.753,43.175,158.316
C08906=1037.898,308.016,380.526,171.749,43.173,158.315
C08907=1037.891,307.769,380.559,171.746,43.172,158.314
C08908=1037.884,307.521,380.593,171.741,43.170,158.313
C08909=1037.877,307.273,380.627,171.737,43.168,158.313
C08910=1037.871,307.026,380.659,171.733,43.166,158.312
C08911=1037.864,306.778,380.693,171.728,43.165,158.311
C08912=1037.856,306.530,380.726,171.724,43.163,158.311
C08913=1037.846,306.172,380.775,171.718,43.161,158.310
C08914=1037.836,305.812,380.823,171.712,43.158,158.309
C08915=1037.826,305.452,380.872,171.707,43.156,158.308
C08916=1037.816,305.093,380.919,171.701,43.154,158.307
C08917=1037.809,304.845,380.952,171.697,43.152,158.306
C08918=1037.802,304.597,380.986,171.692,43.150,158.305
C08919=1037.795,304.349,381.019,171.688,43.149,158.305
C08920=1037.788,304.102,381.053,171.684,43.147,158.304
C08921=1037.781,303.854,381.085,171.680,43.146,158.303
C08922=1037.774,303.607,381.119,171.676,43.144,158.303
C08923=1037.767,303.358,381.152,171.672,43.142,158.302
C08924=1037.761,303.111,381.184,171.668,43.141,158.301
C08925=1037.753,302.864,381.218,171.663,43.139,158.300
C08926=1037.746,302.616,381.250,171.660,43.138,158.300
C08927=1037.739,302.368,381.284,171.656,43.136,158.299
C08928=1037.733,302.121,381.317,171.652,43.134,158.298
C08929=1037.726,301.872,381.350,171.648,43.133,158.298
C08930=1037.719,301.626,381.383,171.643,43.131,158.297
C08931=1037.712,301.377,381.416,171.639,43.130,158.297
C08932=1037.705,301.130,381.449,171.636,43.128,158.296
C08933=1037.699,300.882,381.482,171.632,43.126,158.295
C08934=1037.692,300.635,381.515,171.628,43.124,158.294
C08935=1037.684,300.387,381.548,171.623,43.123,158.294
C08936=1037.678,300.139,381.581,171.619,43.121,158.293
C08937=1037.672,299.891,381.613,171.616,43.120,158.293
C08938=1037.665,299.644,381.647,171.612,43.118,158.292
C08939=1037.658,299.396,381.679,171.608,43.116,158.291
C08940=1037.651,299.148,381.712,171.603,43.115,158.290
C08941=1037.644,298.901,381.745,171.600,43.114,158.290
C08942=1037.638,298.653,381.778,171.596,43.112,158.289
C08943=1037.630,298.405,381.810,171.592,43.111,158.289
C08944=1037.624,298.158,381.844,171.588,43.109,158.288
C08945=1037.617,297.910,381.877,171.585,43.107,158.287
C08946=1037.611,297.662,381.910,171.581,43.105,158.287
C08947=1037.604,297.415,381.942,171.576,43.104,158.286
C08948=1037.597,297.167,381.975,171.572,43.102,158.285
C08949=1037.590,296.919,382.008,171.568,43.101,158.285
C08950=1037.584,296.671,382.041,171.564,43.099,158.284
C08951=1037.576,296.423,382.073,171.561,43.098,158.283
C08952=1037.570,296.176,382.106,171.557,43.097,158.283
C08953=1037.564,295.928,382.139,171.553,43.095,158.282
C08954=1037.558,295.681,382.171,171.550,43.093,158.281
C08955=1037.550,295.433,382.204,171.545,43.092,158.281
C08956=1037.544,295.185,382.237,171.541,43.090,158.280
C08957=1037.537,294.937,382.269,171.537,43.089,158.280
C08958=1037.530,294.689,382.301,171.533,43.087,158.279
C08959=1037.523,294.442,382.333,171.530,43.086,158.278
C08960=1037.517,294.194,382.366,171.526,43.085,158.278
C08961=1037.509,293.946,382.398,171.522,43.083,158.277
C08962=1037.503,293.698,382.431,171.519,43.082,158.277
C08963=1037.496,293.450,382.463,171.515,43.080,158.276
C08964=1037.490,293.203,382.495,171.510,43.079,158.275
C08965=1037.482,292.955,382.528,171.507,43.078,158.275
C08966=1037.475,292.707,382.559,171.503,43.076,158.274
C08967=1037.468,292.460,382.591,171.499,43.075,158.273
C08968=1037.461,292.211,382.625,171.495,43.073,158.273
C08969=1037.452,291.868,382.668,171.490,43.071,158.272
C08970=1037.442,291.526,382.713,171.485,43.070,158.271
C08971=1037.434,291.183,382.757,171.479,43.067,158.270
C08972=1037.424,290.841,382.801,171.474,43.066,158.269
C08973=1037.417,290.592,382.834,171.471,43.064,158.269
C08974=1037.410,290.345,382.866,171.467,43.063,158.268
C08975=1037.403,290.097,382.898,171.463,43.062,158.268
C08976=1037.397,289.849,382.930,171.460,43.060,158.267
C08977=1037.390,289.602,382.962,171.456,43.059,158.267
C08978=1037.383,289.353,382.994,171.452,43.058,158.266
C08979=1037.376,289.106,383.026,171.449,43.056,158.265
C08980=1037.370,288.858,383.058,171.445,43.054,158.265
C08981=1037.363,288.610,383.090,171.441,43.053,158.264
C08982=1037.356,288.362,383.122,171.438,43.052,158.264
C08983=1037.349,288.115,383.153,171.433,43.051,158.263
C08984=1037.342,287.867,383.186,171.429,43.049,158.262
C08985=1037.336,287.618,383.218,171.426,43.048,158.262
C08986=1037.329,287.370,383.249,171.422,43.047,158.261
C08987=1037.322,287.123,383.281,171.418,43.045,158.261
C08988=1037.315,286.875,383.313,171.415,43.044,158.260
C08989=1037.308,286.627,383.344,171.411,43.043,158.260
C08990=1037.302,286.379,383.376,171.407,43.041,158.259
C08991=1037.294,286.132,383.408,171.404,43.041,158.259
C08992=1037.287,285.884,383.440,171.400,43.039,158.258
C08993=1037.281,285.636,383.471,171.396,43.038,158.257
C08994=1037.274,285.388,383.502,171.393,43.037,158.257
C08995=1037.267,285.140,383.534,171.389,43.035,158.256
C08996=1037.260,284.893,383.566,171.385,43.034,158.256
C08997=1037.253,284.645,383.597,171.382,43.033,158.255
C08998=1037.247,284.397,383.629,171.378,43.032,158.255
C08999=1037.240,284.149,383.660,171.375,43.031,158.254
C09000=1037.233,283.900,383.692,171.371,43.030,158.254
C09001=1037.226,283.652,383.724,171.367,43.028,158.253
C09002=1037.219,283.404,383.755,171.364,43.027,158.252
C09003=1037.212,283.157,383.786,171.360,43.026,158.252
C09004=1037.206,282.909,383.818,171.356,43.024,158.251
C09005=1037.199,282.661,383.849,171.353,43.023,158.251
C09006=1037.192,282.413,383.881,171.350,43.022,158.250
C09007=1037.186,282.165,383.912,171.346,43.021,158.250
C09008=1037.179,281.917,383.944,171.343,43.019,158.249
C09009=1037.172,281.669,383.975,171.339,43.018,158.249
C09010=1037.165,281.421,384.006,171.335,43.017,158.248
C09011=1037.159,281.173,384.038,171.332,43.015,158.247
C09012=1037.152,280.925,384.069,171.328,43.015,158.247
C09013=1037.145,280.678,384.101,171.325,43.013,158.246
C09014=1037.138,280.430,384.132,171.321,43.012,158.246
C09015=1037.132,280.182,384.164,171.317,43.011,158.245
C09016=1037.125,279.934,384.195,171.314,43.010,158.245
C09017=1037.118,279.686,384.226,171.310,43.009,158.244
C09018=1037.112,279.437,384.257,171.307,43.007,158.244
C09019=1037.105,279.190,384.289,171.303,43.006,158.243
C09020=1037.099,278.942,384.320,171.300,43.005,158.243
C09021=1037.092,278.694,384.351,171.297,43.004,158.242
C09022=1037.086,278.447,384.383,171.293,43.002,158.242
C09023=1037.078,278.198,384.413,171.289,43.001,158.241
C09024=1037.072,277.950,384.444,171.286,43.000,158.241
C09025=1037.062,277.620,384.485,171.281,42.999,158.240
C09026=1037.054,277.289,384.527,171.276,42.997,158.239
C09027=1037.044,276.958,384.568,171.272,42.996,158.239
C09028=1037.036,276.627,384.610,171.268,42.994,158.238
C09029=1037.029,276.379,384.640,171.264,42.993,158.237
C09030=1037.022,276.131,384.671,171.261,42.992,158.237
C09031=1037.015,275.883,384.703,171.257,42.991,158.236
C09032=1037.008,275.635,384.733,171.253,42.990,158.236
C09033=1037.002,275.387,384.764,171.250,42.988,158.235
C09034=1036.995,275.139,384.796,171.246,42.988,158.235
C09035=1036.988,274.890,384.826,171.243,42.986,158.234
C09036=1036.982,274.644,384.857,171.240,42.985,158.234
C09037=1036.975,274.395,384.888,171.237,42.984,158.233
C09038=1036.968,274.147,384.919,171.233,42.983,158.233
C09039=1036.961,273.899,384.949,171.229,42.982,158.232
C09040=1036.955,273.651,384.981,171.226,42.981,158.232
C09041=1036.948,273.402,385.011,171.222,42.980,158.231
C09042=1036.941,273.156,385.042,171.220,42.979,158.231
C09043=1036.935,272.907,385.072,171.216,42.977,158.230
C09044=1036.927,272.659,385.103,171.213,42.976,158.230
C09045=1036.921,272.411,385.134,171.209,42.975,158.229
C09046=1036.915,272.162,385.165,171.205,42.974,158.229
C09047=1036.908,271.916,385.195,171.202,42.973,158.228
C09048=1036.901,271.667,385.226,171.199,42.972,158.228
C09049=1036.895,271.419,385.257,171.196,42.971,158.227
C09050=1036.887,271.171,385.287,171.192,42.970,158.227
C09051=1036.882,270.923,385.318,171.189,42.969,158.226
C09052=1036.874,270.675,385.348,171.185,42.968,158.226
C09053=1036.868,270.427,385.379,171.182,42.967,158.225
C09054=1036.861,270.179,385.409,171.179,42.966,158.225
C09055=1036.854,269.930,385.440,171.175,42.965,158.224
C09056=1036.848,269.683,385.470,171.172,42.964,158.224
C09057=1036.840,269.435,385.501,171.168,42.963,158.224
C09058=1036.834,269.187,385.531,171.166,42.962,158.223
C09059=1036.827,268.939,385.561,171.162,42.961,158.223
C09060=1036.821,268.691,385.592,171.159,42.960,158.222
C09061=1036.814,268.442,385.622,171.155,42.959,158.222
C09062=1036.807,268.194,385.654,171.152,42.957,158.221
C09063=1036.800,267.947,385.683,171.149,42.957,158.221
C09064=1036.794,267.698,385.714,171.146,42.956,158.220
C09065=1036.787,267.450,385.744,171.142,42.955,158.220
C09066=1036.780,267.203,385.774,171.138,42.954,158.219
C09067=1036.774,266.954,385.805,171.136,42.952,158.219
C09068=1036.767,266.706,385.835,171.132,42.952,158.218
C09069=1036.760,266.458,385.864,171.129,42.951,158.218
C09070=1036.754,266.210,385.895,171.125,42.950,158.217
C09071=1036.746,265.962,385.925,171.122,42.949,158.217
C09072=1036.739,265.713,385.955,171.119,42.948,158.217
C09073=1036.733,265.466,385.986,171.116,42.947,158.216
C09074=1036.726,265.217,386.016,171.112,42.946,158.216
C09075=1036.720,264.970,386.046,171.109,42.945,158.215
C09076=1036.713,264.721,386.076,171.106,42.944,158.215
C09077=1036.706,264.473,386.107,171.103,42.943,158.214
C09078=1036.700,264.226,386.136,171.099,42.942,158.214
C09079=1036.692,263.977,386.166,171.097,42.941,158.213
C09080=1036.686,263.729,386.197,171.093,42.940,158.213
C09081=1036.677,263.403,386.236,171.088,42.939,158.212
C09082=1036.669,263.077,386.275,171.085,42.937,158.212
C09083=1036.660,262.750,386.315,171.080,42.936,158.211
C09084=1036.651,262.425,386.355,171.076,42.935,158.211
C09085=1036.644,262.176,386.384,171.073,42.934,158.210
C09086=1036.638,261.928,386.414,171.070,42.933,158.210
C09087=1036.632,261.680,386.445,171.067,42.932,158.209
C09088=1036.624,261.431,386.475,171.063,42.931,158.209
C09089=1036.617,261.184,386.503,171.060,42.930,158.208
C09090=1036.610,260.935,386.533,171.057,42.930,158.208
C09091=1036.603,260.687,386.563,171.054,42.929,158.208
C09092=1036.597,260.439,386.593,171.051,42.928,158.207
C09093=1036.590,260.191,386.623,171.047,42.927,158.207
C09094=1036.583,259.943,386.652,171.044,42.926,158.206
C09095=1036.576,259.695,386.682,171.041,42.925,158.206
C09096=1036.569,259.446,386.712,171.038,42.924,158.205
C09097=1036.563,259.198,386.741,171.034,42.924,158.205
C09098=1036.556,258.950,386.771,171.032,42.923,158.205
C09099=1036.549,258.702,386.800,171.028,42.922,158.204
C09100=1036.542,258.454,386.830,171.025,42.921,158.204
C09101=1036.535,258.206,386.859,171.021,42.921,158.203
C09102=1036.528,257.958,386.889,171.019,42.920,158.203
C09103=1036.522,257.710,386.918,171.016,42.919,158.203
C09104=1036.515,257.461,386.948,171.012,42.918,158.202
C09105=1036.508,257.213,386.977,171.009,42.917,158.202
